KUKA KRL program: MyProgram_008().src

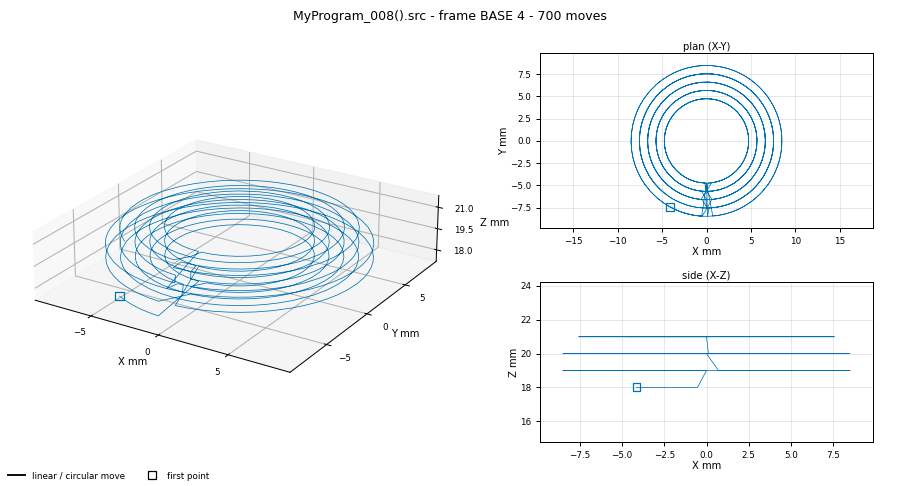
[picture p0: tool path of MyProgram_008().src in frame BASE 4, 700 of 700 moves have a stored position in this frame; points joined in program order, loops and branches not executed]
&ACCESS RVP
&REL 1
&PARAM TEMPLATE = C:\KRC\Roboter\Template\vorgabe
&PARAM EDITMASK = *
DEF MyProgram_008()
; ---- Setting reference (Base) ----
$BASE = BASE_DATA[4]

; --------------------------
; ---- Setting tool (TCP) ----
$TOOL = TOOL_DATA[3]
; --------------------------

$VEL.CP = VEL_APROX_PRINT
Startdeposition()
$VEL.CP = VEL_PRINT
LIN {X -4.1408,Y -7.4105,Z 18,A -3.2305,B 0,C 0,E1 0.1598,E2 90.0712} C_DIS
LIN {X -3.4628,Y -7.7493,Z 18,A -3.22,B 0,C 0,E1 0.1598,E2 90.0712} C_DIS
LIN {X -2.7578,Y -8.0269,Z 18,A -3.2059,B 0,C 0,E1 0.1598,E2 90.0712} C_DIS
LIN {X -2.031,Y -8.2415,Z 18,A -3.1884,B 0,C 0,E1 0.1598,E2 90.0712} C_DIS
LIN {X -1.288,Y -8.391,Z 18,A -3.1675,B 0,C 0,E1 0.1598,E2 90.0713} C_DIS
LIN {X -0.5343,Y -8.4709,Z 18,A -3.1433,B 0,C 0,E1 0.1598,E2 90.0713} C_DIS
LIN {X -0.5343,Y -8.4709,Z 18,A -3.1433,B 0,C 0,E1 0.1598,E2 90.0713} C_DIS
Enddeposition()
LIN {X 0.0003,Y -4.7568,Z 19,A -2.951,B 0,C 0,E1 0.1598,E2 90.0603} C_DIS
Startdeposition()
$VEL.CP = VEL_PRINT
LIN {X 0.0003,Y -4.7568,Z 19,A -2.9567,B 0,C 0,E1 0.1598,E2 90.0661} C_DIS
LIN {X -0.9266,Y -4.6606,Z 19,A -2.9915,B 0,C 0,E1 0.1598,E2 90.0709} C_DIS
LIN {X -1.6437,Y -4.457,Z 19,A -3.0098,B 0,C 0,E1 0.1598,E2 90.0715} C_DIS
LIN {X -2.3205,Y -4.1449,Z 19,A -3.0215,B 0,C 0,E1 0.1598,E2 90.0715} C_DIS
LIN {X -2.9394,Y -3.7297,Z 19,A -3.0266,B 0,C 0,E1 0.1598,E2 90.0715} C_DIS
LIN {X -3.4873,Y -3.2244,Z 19,A -3.0253,B 0,C 0,E1 0.1598,E2 90.0714} C_DIS
LIN {X -3.9485,Y -2.6389,Z 19,A -3.0174,B 0,C 0,E1 0.1598,E2 90.0714} C_DIS
LIN {X -4.314,Y -1.9893,Z 19,A -3.0034,B 0,C 0,E1 0.1598,E2 90.0714} C_DIS
LIN {X -4.5707,Y -1.2895,Z 19,A -2.9832,B 0,C 0,E1 0.1598,E2 90.0714} C_DIS
LIN {X -4.716,Y -0.5586,Z 19,A -2.9577,B 0,C 0,E1 0.1598,E2 90.0714} C_DIS
LIN {X -4.7458,Y 0.1861,Z 19,A -2.9273,B 0,C 0,E1 0.1598,E2 90.0714} C_DIS
LIN {X -4.6607,Y 0.9267,Z 19,A -2.8929,B 0,C 0,E1 0.1598,E2 90.0714} C_DIS
LIN {X -4.4566,Y 1.6437,Z 19,A -2.8551,B 0,C 0,E1 0.1598,E2 90.0715} C_DIS
LIN {X -4.1446,Y 2.3207,Z 19,A -2.8151,B 0,C 0,E1 0.1598,E2 90.0715} C_DIS
LIN {X -3.7315,Y 2.9411,Z 19,A -2.7737,B 0,C 0,E1 0.1598,E2 90.0717} C_DIS
LIN {X -3.225,Y 3.4882,Z 19,A -2.732,B 0,C 0,E1 0.1598,E2 90.0717} C_DIS
LIN {X -2.6388,Y 3.9486,Z 19,A -2.691,B 0,C 0,E1 0.1598,E2 90.0719} C_DIS
LIN {X -1.9887,Y 4.313,Z 19,A -2.6517,B 0,C 0,E1 0.1598,E2 90.0719} C_DIS
LIN {X -1.1995,Y 4.5956,Z 19,A -2.6107,B 0,C 0,E1 0.1598,E2 90.0721} C_DIS
LIN {X -0.5587,Y 4.7185,Z 19,A -2.5819,B 0,C 0,E1 0.1598,E2 90.0721} C_DIS
LIN {X 0.1862,Y 4.749,Z 19,A -2.5532,B 0,C 0,E1 0.1598,E2 90.0721} C_DIS
LIN {X 0.9266,Y 4.6606,Z 19,A -2.5296,B 0,C 0,E1 0.1598,E2 90.0721} C_DIS
LIN {X 1.6433,Y 4.456,Z 19,A -2.5118,B 0,C 0,E1 0.1598,E2 90.0721} C_DIS
LIN {X 2.3206,Y 4.1447,Z 19,A -2.5,B 0,C 0,E1 0.1598,E2 90.0721} C_DIS
LIN {X 2.9416,Y 3.7322,Z 19,A -2.4945,B 0,C 0,E1 0.1598,E2 90.0721} C_DIS
LIN {X 3.4881,Y 3.2248,Z 19,A -2.4958,B 0,C 0,E1 0.1598,E2 90.0721} C_DIS
LIN {X 3.9509,Y 2.6404,Z 19,A -2.5035,B 0,C 0,E1 0.1598,E2 90.0721} C_DIS
LIN {X 4.3138,Y 1.989,Z 19,A -2.5177,B 0,C 0,E1 0.1598,E2 90.072} C_DIS
LIN {X 4.5707,Y 1.2894,Z 19,A -2.5379,B 0,C 0,E1 0.1598,E2 90.072} C_DIS
LIN {X 4.7184,Y 0.5588,Z 19,A -2.5635,B 0,C 0,E1 0.1598,E2 90.0719} C_DIS
LIN {X 4.7489,Y -0.1862,Z 19,A -2.594,B 0,C 0,E1 0.1598,E2 90.0719} C_DIS
LIN {X 4.6591,Y -0.9263,Z 19,A -2.6287,B 0,C 0,E1 0.1598,E2 90.0718} C_DIS
LIN {X 4.4556,Y -1.6435,Z 19,A -2.6666,B 0,C 0,E1 0.1598,E2 90.0718} C_DIS
LIN {X 4.1448,Y -2.3207,Z 19,A -2.7068,B 0,C 0,E1 0.1598,E2 90.0718} C_DIS
LIN {X 3.7299,Y -2.9399,Z 19,A -2.7484,B 0,C 0,E1 0.1598,E2 90.0718} C_DIS
LIN {X 3.2242,Y -3.4874,Z 19,A -2.7903,B 0,C 0,E1 0.1598,E2 90.0718} C_DIS
LIN {X 2.6388,Y -3.9486,Z 19,A -2.8314,B 0,C 0,E1 0.1598,E2 90.0717} C_DIS
LIN {X 1.9887,Y -4.313,Z 19,A -2.8708,B 0,C 0,E1 0.1598,E2 90.0717} C_DIS
LIN {X 1.1996,Y -4.5956,Z 19,A -2.9118,B 0,C 0,E1 0.1598,E2 90.0717} C_DIS
LIN {X 0.5588,Y -4.7187,Z 19,A -2.9405,B 0,C 0,E1 0.1598,E2 90.0717} C_DIS
LIN {X 0.5588,Y -4.7187,Z 19,A -2.9405,B 0,C 0,E1 0.1598,E2 90.0717} C_DIS
Enddeposition()
LIN {X 0,Y -5.6862,Z 19,A -3.001,B 0,C 0,E1 0.1598,E2 90.0704} C_DIS
Startdeposition()
$VEL.CP = VEL_PRINT
LIN {X 0.6409,Y -5.6452,Z 19,A -2.9769,B 0,C 0,E1 0.1598,E2 90.0715} C_DIS
LIN {X 1.4817,Y -5.4861,Z 19,A -2.9393,B 0,C 0,E1 0.1598,E2 90.0716} C_DIS
LIN {X 2.2884,Y -5.2009,Z 19,A -2.8976,B 0,C 0,E1 0.1598,E2 90.0716} C_DIS
LIN {X 3.0434,Y -4.7981,Z 19,A -2.8527,B 0,C 0,E1 0.1598,E2 90.0716} C_DIS
LIN {X 3.7291,Y -4.2862,Z 19,A -2.8058,B 0,C 0,E1 0.1598,E2 90.0717} C_DIS
LIN {X 4.3305,Y -3.6775,Z 19,A -2.7578,B 0,C 0,E1 0.1598,E2 90.0717} C_DIS
LIN {X 4.8347,Y -2.986,Z 19,A -2.7098,B 0,C 0,E1 0.1598,E2 90.0717} C_DIS
LIN {X 5.2278,Y -2.226,Z 19,A -2.663,B 0,C 0,E1 0.1598,E2 90.0717} C_DIS
LIN {X 5.5023,Y -1.4156,Z 19,A -2.6184,B 0,C 0,E1 0.1598,E2 90.0717} C_DIS
LIN {X 5.6534,Y -0.5733,Z 19,A -2.5771,B 0,C 0,E1 0.1598,E2 90.0717} C_DIS
LIN {X 5.6763,Y 0.2822,Z 19,A -2.5399,B 0,C 0,E1 0.1598,E2 90.0717} C_DIS
LIN {X 5.5702,Y 1.1315,Z 19,A -2.5077,B 0,C 0,E1 0.1598,E2 90.0718} C_DIS
LIN {X 5.3355,Y 1.9546,Z 19,A -2.4814,B 0,C 0,E1 0.1598,E2 90.0718} C_DIS
LIN {X 4.9812,Y 2.7335,Z 19,A -2.4614,B 0,C 0,E1 0.1598,E2 90.0719} C_DIS
LIN {X 4.514,Y 3.4505,Z 19,A -2.4483,B 0,C 0,E1 0.1598,E2 90.072} C_DIS
LIN {X 3.945,Y 4.0897,Z 19,A -2.4422,B 0,C 0,E1 0.1598,E2 90.072} C_DIS
LIN {X 3.2863,Y 4.6361,Z 19,A -2.4434,B 0,C 0,E1 0.1598,E2 90.0721} C_DIS
LIN {X 2.5533,Y 5.0782,Z 19,A -2.4518,B 0,C 0,E1 0.1598,E2 90.0721} C_DIS
LIN {X 1.7619,Y 5.4046,Z 19,A -2.4672,B 0,C 0,E1 0.1598,E2 90.0722} C_DIS
LIN {X 0.9303,Y 5.6086,Z 19,A -2.4893,B 0,C 0,E1 0.1598,E2 90.0722} C_DIS
LIN {X 0.0776,Y 5.6849,Z 19,A -2.5175,B 0,C 0,E1 0.1598,E2 90.0722} C_DIS
LIN {X -0.7768,Y 5.6314,Z 19,A -2.5513,B 0,C 0,E1 0.1598,E2 90.0722} C_DIS
LIN {X -1.614,Y 5.4516,Z 19,A -2.5898,B 0,C 0,E1 0.1598,E2 90.0722} C_DIS
LIN {X -2.4546,Y 5.1327,Z 19,A -2.6342,B 0,C 0,E1 0.1598,E2 90.072} C_DIS
LIN {X -3.5239,Y 4.4596,Z 19,A -2.7019,B 0,C 0,E1 0.1598,E2 90.0718} C_DIS
LIN {X -4.0794,Y 3.9571,Z 19,A -2.7436,B 0,C 0,E1 0.1598,E2 90.0718} C_DIS
LIN {X -4.5642,Y 3.3862,Z 19,A -2.7855,B 0,C 0,E1 0.1598,E2 90.0717} C_DIS
LIN {X -4.9699,Y 2.7566,Z 19,A -2.827,B 0,C 0,E1 0.1598,E2 90.0717} C_DIS
LIN {X -5.2905,Y 2.0796,Z 19,A -2.8673,B 0,C 0,E1 0.1598,E2 90.0715} C_DIS
LIN {X -5.5194,Y 1.3661,Z 19,A -2.9058,B 0,C 0,E1 0.1598,E2 90.0715} C_DIS
LIN {X -5.6499,Y 0.6283,Z 19,A -2.9417,B 0,C 0,E1 0.1598,E2 90.0714} C_DIS
LIN {X -5.6842,Y -0.12,Z 19,A -2.9746,B 0,C 0,E1 0.1598,E2 90.0714} C_DIS
LIN {X -5.6165,Y -0.8662,Z 19,A -3.0036,B 0,C 0,E1 0.1598,E2 90.0713} C_DIS
LIN {X -5.4547,Y -1.5974,Z 19,A -3.0285,B 0,C 0,E1 0.1598,E2 90.0713} C_DIS
LIN {X -5.1973,Y -2.3009,Z 19,A -3.0488,B 0,C 0,E1 0.1598,E2 90.0713} C_DIS
LIN {X -4.8517,Y -2.9656,Z 19,A -3.0642,B 0,C 0,E1 0.1598,E2 90.0713} C_DIS
LIN {X -4.4183,Y -3.5769,Z 19,A -3.0741,B 0,C 0,E1 0.1598,E2 90.0713} C_DIS
LIN {X -3.9082,Y -4.1255,Z 19,A -3.0786,B 0,C 0,E1 0.1598,E2 90.0713} C_DIS
LIN {X -3.3325,Y -4.6046,Z 19,A -3.0778,B 0,C 0,E1 0.1598,E2 90.0713} C_DIS
LIN {X -2.6973,Y -5.0015,Z 19,A -3.0713,B 0,C 0,E1 0.1598,E2 90.0713} C_DIS
LIN {X -2.0167,Y -5.3143,Z 19,A -3.0596,B 0,C 0,E1 0.1598,E2 90.0714} C_DIS
LIN {X -1.3007,Y -5.5351,Z 19,A -3.0427,B 0,C 0,E1 0.1598,E2 90.0714} C_DIS
LIN {X -0.5612,Y -5.6557,Z 19,A -3.0207,B 0,C 0,E1 0.1598,E2 90.0715} C_DIS
LIN {X -0.5612,Y -5.6557,Z 19,A -3.0207,B 0,C 0,E1 0.1598,E2 90.0715} C_DIS
Enddeposition()
LIN {X 0.0261,Y -6.6218,Z 19,A -3.0391,B 0,C 0,E1 0.1598,E2 90.0703} C_DIS
Startdeposition()
$VEL.CP = VEL_PRINT
LIN {X -0.8856,Y -6.5586,Z 19,A -3.0709,B 0,C 0,E1 0.1598,E2 90.0714} C_DIS
LIN {X -1.6037,Y -6.4211,Z 19,A -3.0915,B 0,C 0,E1 0.1598,E2 90.0714} C_DIS
LIN {X -2.3028,Y -6.2069,Z 19,A -3.1081,B 0,C 0,E1 0.1598,E2 90.0714} C_DIS
LIN {X -2.9723,Y -5.9126,Z 19,A -3.1201,B 0,C 0,E1 0.1598,E2 90.0714} C_DIS
LIN {X -3.607,Y -5.5497,Z 19,A -3.1281,B 0,C 0,E1 0.1598,E2 90.0714} C_DIS
LIN {X -4.1979,Y -5.1188,Z 19,A -3.1315,B 0,C 0,E1 0.1598,E2 90.0713} C_DIS
LIN {X -4.7363,Y -4.6238,Z 19,A -3.1303,B 0,C 0,E1 0.1598,E2 90.0713} C_DIS
LIN {X -5.217,Y -4.0727,Z 19,A -3.1246,B 0,C 0,E1 0.1598,E2 90.0713} C_DIS
LIN {X -5.6344,Y -3.4723,Z 19,A -3.1145,B 0,C 0,E1 0.1598,E2 90.0713} C_DIS
LIN {X -5.9829,Y -2.8295,Z 19,A -3.1002,B 0,C 0,E1 0.1598,E2 90.0713} C_DIS
LIN {X -6.2578,Y -2.1521,Z 19,A -3.0817,B 0,C 0,E1 0.1598,E2 90.0713} C_DIS
LIN {X -6.4587,Y -1.449,Z 19,A -3.0593,B 0,C 0,E1 0.1598,E2 90.0713} C_DIS
LIN {X -6.5806,Y -0.7279,Z 19,A -3.0334,B 0,C 0,E1 0.1598,E2 90.0713} C_DIS
LIN {X -6.6194,Y 0.0024,Z 19,A -3.004,B 0,C 0,E1 0.1598,E2 90.0713} C_DIS
LIN {X -6.5797,Y 0.7325,Z 19,A -2.9717,B 0,C 0,E1 0.1598,E2 90.0713} C_DIS
LIN {X -6.4575,Y 1.4535,Z 19,A -2.9368,B 0,C 0,E1 0.1598,E2 90.0713} C_DIS
LIN {X -6.2582,Y 2.1571,Z 19,A -2.8999,B 0,C 0,E1 0.1598,E2 90.0715} C_DIS
LIN {X -5.9836,Y 2.8348,Z 19,A -2.8612,B 0,C 0,E1 0.1598,E2 90.0715} C_DIS
LIN {X -5.6316,Y 3.4757,Z 19,A -2.8212,B 0,C 0,E1 0.1598,E2 90.0716} C_DIS
LIN {X -5.2138,Y 4.0758,Z 19,A -2.7805,B 0,C 0,E1 0.1598,E2 90.0716} C_DIS
LIN {X -4.7331,Y 4.6268,Z 19,A -2.7396,B 0,C 0,E1 0.1598,E2 90.0718} C_DIS
LIN {X -4.195,Y 5.1216,Z 19,A -2.6989,B 0,C 0,E1 0.1598,E2 90.0718} C_DIS
LIN {X -3.6043,Y 5.5527,Z 19,A -2.659,B 0,C 0,E1 0.1598,E2 90.0719} C_DIS
LIN {X -2.97,Y 5.9168,Z 19,A -2.6202,B 0,C 0,E1 0.1598,E2 90.072} C_DIS
LIN {X -2.2998,Y 6.2097,Z 19,A -2.5832,B 0,C 0,E1 0.1598,E2 90.072} C_DIS
LIN {X -1.6007,Y 6.4242,Z 19,A -2.5483,B 0,C 0,E1 0.1598,E2 90.0722} C_DIS
LIN {X -0.701,Y 6.5862,Z 19,A -2.5083,B 0,C 0,E1 0.1598,E2 90.0722} C_DIS
LIN {X 0.455,Y 6.6038,Z 19,A -2.4649,B 0,C 0,E1 0.1598,E2 90.0722} C_DIS
LIN {X 1.6036,Y 6.4264,Z 19,A -2.43,B 0,C 0,E1 0.1598,E2 90.0723} C_DIS
LIN {X 2.5114,Y 6.1237,Z 19,A -2.4093,B 0,C 0,E1 0.1598,E2 90.0723} C_DIS
LIN {X 3.2013,Y 5.7918,Z 19,A -2.3979,B 0,C 0,E1 0.1598,E2 90.0723} C_DIS
LIN {X 3.849,Y 5.3838,Z 19,A -2.3913,B 0,C 0,E1 0.1598,E2 90.0723} C_DIS
LIN {X 4.4444,Y 4.9029,Z 19,A -2.3896,B 0,C 0,E1 0.1598,E2 90.0723} C_DIS
LIN {X 4.9809,Y 4.357,Z 19,A -2.393,B 0,C 0,E1 0.1598,E2 90.0722} C_DIS
LIN {X 5.4509,Y 3.7528,Z 19,A -2.4012,B 0,C 0,E1 0.1598,E2 90.0722} C_DIS
LIN {X 5.8483,Y 3.0985,Z 19,A -2.4143,B 0,C 0,E1 0.1598,E2 90.0721} C_DIS
LIN {X 6.1677,Y 2.4028,Z 19,A -2.4321,B 0,C 0,E1 0.1598,E2 90.0721} C_DIS
LIN {X 6.4042,Y 1.6746,Z 19,A -2.4542,B 0,C 0,E1 0.1598,E2 90.072} C_DIS
LIN {X 6.5537,Y 0.9237,Z 19,A -2.4806,B 0,C 0,E1 0.1598,E2 90.072} C_DIS
LIN {X 6.6156,Y 0.1609,Z 19,A -2.5107,B 0,C 0,E1 0.1598,E2 90.0719} C_DIS
LIN {X 6.5914,Y -0.6042,Z 19,A -2.5441,B 0,C 0,E1 0.1598,E2 90.0719} C_DIS
LIN {X 6.4774,Y -1.3612,Z 19,A -2.5805,B 0,C 0,E1 0.1598,E2 90.0719} C_DIS
LIN {X 6.2764,Y -2.0999,Z 19,A -2.6193,B 0,C 0,E1 0.1598,E2 90.0718} C_DIS
LIN {X 5.9941,Y -2.8114,Z 19,A -2.66,B 0,C 0,E1 0.1598,E2 90.0718} C_DIS
LIN {X 5.6304,Y -3.4851,Z 19,A -2.702,B 0,C 0,E1 0.1598,E2 90.0718} C_DIS
LIN {X 5.1873,Y -4.1094,Z 19,A -2.7448,B 0,C 0,E1 0.1598,E2 90.0718} C_DIS
LIN {X 4.6785,Y -4.6812,Z 19,A -2.7878,B 0,C 0,E1 0.1598,E2 90.0717} C_DIS
LIN {X 4.1066,Y -5.19,Z 19,A -2.8305,B 0,C 0,E1 0.1598,E2 90.0717} C_DIS
LIN {X 3.4797,Y -5.6294,Z 19,A -2.8722,B 0,C 0,E1 0.1598,E2 90.0717} C_DIS
LIN {X 2.8072,Y -5.9951,Z 19,A -2.9124,B 0,C 0,E1 0.1598,E2 90.0717} C_DIS
LIN {X 2.0961,Y -6.2792,Z 19,A -2.9506,B 0,C 0,E1 0.1598,E2 90.0717} C_DIS
LIN {X 1.3572,Y -6.4796,Z 19,A -2.9862,B 0,C 0,E1 0.1598,E2 90.0716} C_DIS
LIN {X 0.5998,Y -6.5922,Z 19,A -3.0188,B 0,C 0,E1 0.1598,E2 90.0716} C_DIS
LIN {X 0.5998,Y -6.5922,Z 19,A -3.0188,B 0,C 0,E1 0.1598,E2 90.0716} C_DIS
Enddeposition()
LIN {X 0.0596,Y -7.5563,Z 19,A -3.0785,B 0,C 0,E1 0.1598,E2 90.0703} C_DIS
Startdeposition()
$VEL.CP = VEL_PRINT
LIN {X 0.9093,Y -7.5022,Z 19,A -3.0462,B 0,C 0,E1 0.1598,E2 90.0715} C_DIS
LIN {X 2.0403,Y -7.2731,Z 19,A -2.995,B 0,C 0,E1 0.1598,E2 90.0715} C_DIS
LIN {X 2.9949,Y -6.9378,Z 19,A -2.9457,B 0,C 0,E1 0.1598,E2 90.0715} C_DIS
LIN {X 3.9106,Y -6.4663,Z 19,A -2.8921,B 0,C 0,E1 0.1598,E2 90.0716} C_DIS
LIN {X 4.6992,Y -5.9141,Z 19,A -2.8396,B 0,C 0,E1 0.1598,E2 90.0716} C_DIS
LIN {X 5.276,Y -5.4037,Z 19,A -2.7968,B 0,C 0,E1 0.1598,E2 90.0717} C_DIS
LIN {X 5.7989,Y -4.8384,Z 19,A -2.7535,B 0,C 0,E1 0.1598,E2 90.0717} C_DIS
LIN {X 6.3712,Y -4.0643,Z 19,A -2.6994,B 0,C 0,E1 0.1598,E2 90.0717} C_DIS
LIN {X 7.0456,Y -2.735,Z 19,A -2.6176,B 0,C 0,E1 0.1598,E2 90.0712} C_DIS
LIN {X 7.3713,Y -1.6678,Z 19,A -2.5604,B 0,C 0,E1 0.1598,E2 90.0715} C_DIS
LIN {X 7.5325,Y -0.6167,Z 19,A -2.5098,B 0,C 0,E1 0.1598,E2 90.0716} C_DIS
LIN {X 7.5419,Y 0.4018,Z 19,A -2.4662,B 0,C 0,E1 0.1598,E2 90.0717} C_DIS
LIN {X 7.4027,Y 1.5186,Z 19,A -2.4237,B 0,C 0,E1 0.1598,E2 90.0717} C_DIS
LIN {X 7.1897,Y 2.3275,Z 19,A -2.3975,B 0,C 0,E1 0.1598,E2 90.072} C_DIS
LIN {X 6.7449,Y 3.4003,Z 19,A -2.368,B 0,C 0,E1 0.1598,E2 90.0717} C_DIS
LIN {X 6.342,Y 4.1018,Z 19,A -2.3534,B 0,C 0,E1 0.1598,E2 90.0721} C_DIS
LIN {X 5.8671,Y 4.7568,Z 19,A -2.3432,B 0,C 0,E1 0.1598,E2 90.0721} C_DIS
LIN {X 5.3248,Y 5.3573,Z 19,A -2.3378,B 0,C 0,E1 0.1598,E2 90.0722} C_DIS
LIN {X 4.5636,Y 6.023,Z 19,A -2.3375,B 0,C 0,E1 0.1598,E2 90.0722} C_DIS
LIN {X 3.61,Y 6.635,Z 19,A -2.3468,B 0,C 0,E1 0.1598,E2 90.0722} C_DIS
LIN {X 2.6664,Y 7.0708,Z 19,A -2.3633,B 0,C 0,E1 0.1598,E2 90.0722} C_DIS
LIN {X 1.6408,Y 7.377,Z 19,A -2.3883,B 0,C 0,E1 0.1598,E2 90.0723} C_DIS
LIN {X 0.7499,Y 7.5202,Z 19,A -2.4152,B 0,C 0,E1 0.1598,E2 90.0723} C_DIS
LIN {X -0.2197,Y 7.5539,Z 19,A -2.4496,B 0,C 0,E1 0.1598,E2 90.0723} C_DIS
LIN {X -1.2608,Y 7.4511,Z 19,A -2.4923,B 0,C 0,E1 0.1598,E2 90.0723} C_DIS
LIN {X -2.3419,Y 7.1807,Z 19,A -2.5436,B 0,C 0,E1 0.1598,E2 90.0722} C_DIS
LIN {X -3.1716,Y 6.8543,Z 19,A -2.588,B 0,C 0,E1 0.1598,E2 90.0721} C_DIS
LIN {X -3.9585,Y 6.4347,Z 19,A -2.6347,B 0,C 0,E1 0.1598,E2 90.072} C_DIS
LIN {X -4.9384,Y 5.7195,Z 19,A -2.7009,B 0,C 0,E1 0.1598,E2 90.0717} C_DIS
LIN {X -5.6771,Y 4.9879,Z 19,A -2.7589,B 0,C 0,E1 0.1598,E2 90.0717} C_DIS
LIN {X -6.2659,Y 4.2161,Z 19,A -2.8131,B 0,C 0,E1 0.1598,E2 90.0716} C_DIS
LIN {X -6.759,Y 3.38,Z 19,A -2.8664,B 0,C 0,E1 0.1598,E2 90.0713} C_DIS
LIN {X -7.2749,Y 2.0498,Z 19,A -2.9409,B 0,C 0,E1 0.1598,E2 90.0707} C_DIS
LIN {X -7.5164,Y 0.7835,Z 19,A -3.0033,B 0,C 0,E1 0.1598,E2 90.0707} C_DIS
LIN {X -7.5569,Y -0.0876,Z 19,A -3.0419,B 0,C 0,E1 0.1598,E2 90.0711} C_DIS
LIN {X -7.4292,Y -1.3623,Z 19,A -3.0904,B 0,C 0,E1 0.1598,E2 90.0706} C_DIS
LIN {X -7.2654,Y -2.0847,Z 19,A -3.1154,B 0,C 0,E1 0.1598,E2 90.071} C_DIS
LIN {X -6.861,Y -3.158,Z 19,A -3.1457,B 0,C 0,E1 0.1598,E2 90.0708} C_DIS
LIN {X -6.2752,Y -4.2109,Z 19,A -3.1686,B 0,C 0,E1 0.1598,E2 90.0708} C_DIS
LIN {X -5.7777,Y -4.8704,Z 19,A -3.1784,B 0,C 0,E1 0.1598,E2 90.071} C_DIS
LIN {X -5.079,Y -5.5909,Z 19,A -3.1833,B 0,C 0,E1 0.1598,E2 90.071} C_DIS
LIN {X -4.4563,Y -6.0978,Z 19,A -3.182,B 0,C 0,E1 0.1598,E2 90.0712} C_DIS
LIN {X -3.7835,Y -6.5358,Z 19,A -3.1759,B 0,C 0,E1 0.1598,E2 90.0712} C_DIS
LIN {X -3.0689,Y -6.9019,Z 19,A -3.1652,B 0,C 0,E1 0.1598,E2 90.0712} C_DIS
LIN {X -1.9814,Y -7.2927,Z 19,A -3.1418,B 0,C 0,E1 0.1598,E2 90.0713} C_DIS
LIN {X -0.9532,Y -7.4972,Z 19,A -3.1129,B 0,C 0,E1 0.1598,E2 90.0713} C_DIS
LIN {X 0.0596,Y -7.5563,Z 19,A -3.0782,B 0,C 0,E1 0.1598,E2 90.0715} C_DIS
Enddeposition()
LIN {X 0.0596,Y -7.5563,Z 19,A -3.0782,B 0,C 0,E1 0.1598,E2 90.0715} C_DIS
Startdeposition()
$VEL.CP = VEL_PRINT
LIN {X -0.4894,Y -8.4742,Z 19,A -3.137,B 0,C 0,E1 0.1598,E2 90.0708} C_DIS
LIN {X -1.2506,Y -8.3958,Z 19,A -3.162,B 0,C 0,E1 0.1598,E2 90.0713} C_DIS
LIN {X -2.0013,Y -8.2484,Z 19,A -3.1833,B 0,C 0,E1 0.1598,E2 90.0713} C_DIS
LIN {X -2.7359,Y -8.0344,Z 19,A -3.2012,B 0,C 0,E1 0.1598,E2 90.0713} C_DIS
LIN {X -3.4483,Y -7.7557,Z 19,A -3.2155,B 0,C 0,E1 0.1598,E2 90.0713} C_DIS
LIN {X -4.1333,Y -7.4148,Z 19,A -3.2261,B 0,C 0,E1 0.1598,E2 90.0713} C_DIS
LIN {X -4.7837,Y -7.0118,Z 19,A -3.2329,B 0,C 0,E1 0.1598,E2 90.0712} C_DIS
LIN {X -5.5434,Y -6.4306,Z 19,A -3.2361,B 0,C 0,E1 0.1598,E2 90.071} C_DIS
LIN {X -6.3513,Y -5.6359,Z 19,A -3.232,B 0,C 0,E1 0.1598,E2 90.071} C_DIS
LIN {X -6.9717,Y -4.8405,Z 19,A -3.2212,B 0,C 0,E1 0.1598,E2 90.071} C_DIS
LIN {X -7.3989,Y -4.1558,Z 19,A -3.208,B 0,C 0,E1 0.1598,E2 90.071} C_DIS
LIN {X -7.7607,Y -3.4345,Z 19,A -3.1909,B 0,C 0,E1 0.1598,E2 90.071} C_DIS
LIN {X -8.0526,Y -2.682,Z 19,A -3.1698,B 0,C 0,E1 0.1598,E2 90.071} C_DIS
LIN {X -8.2711,Y -1.905,Z 19,A -3.1451,B 0,C 0,E1 0.1598,E2 90.071} C_DIS
LIN {X -8.4144,Y -1.1108,Z 19,A -3.1168,B 0,C 0,E1 0.1598,E2 90.071} C_DIS
LIN {X -8.4903,Y -0.1049,Z 19,A -3.077,B 0,C 0,E1 0.1598,E2 90.0709} C_DIS
LIN {X -8.4259,Y 1.0155,Z 19,A -3.0273,B 0,C 0,E1 0.1598,E2 90.0709} C_DIS
LIN {X -8.2936,Y 1.8064,Z 19,A -2.9895,B 0,C 0,E1 0.1598,E2 90.0713} C_DIS
LIN {X -8.0861,Y 2.581,Z 19,A -2.9492,B 0,C 0,E1 0.1598,E2 90.0713} C_DIS
LIN {X -7.8078,Y 3.3331,Z 19,A -2.9073,B 0,C 0,E1 0.1598,E2 90.0714} C_DIS
LIN {X -7.4578,Y 4.0548,Z 19,A -2.864,B 0,C 0,E1 0.1598,E2 90.0714} C_DIS
LIN {X -7.041,Y 4.7398,Z 19,A -2.8198,B 0,C 0,E1 0.1598,E2 90.0716} C_DIS
LIN {X -6.4349,Y 5.5383,Z 19,A -2.7637,B 0,C 0,E1 0.1598,E2 90.0716} C_DIS
LIN {X -5.6183,Y 6.3622,Z 19,A -2.6989,B 0,C 0,E1 0.1598,E2 90.0716} C_DIS
LIN {X -4.9802,Y 6.8722,Z 19,A -2.6541,B 0,C 0,E1 0.1598,E2 90.0719} C_DIS
LIN {X -4.2961,Y 7.3187,Z 19,A -2.61,B 0,C 0,E1 0.1598,E2 90.0719} C_DIS
LIN {X -3.5723,Y 7.6974,Z 19,A -2.5674,B 0,C 0,E1 0.1598,E2 90.0721} C_DIS
LIN {X -2.8157,Y 8.005,Z 19,A -2.5265,B 0,C 0,E1 0.1598,E2 90.0721} C_DIS
LIN {X -2.033,Y 8.2385,Z 19,A -2.4878,B 0,C 0,E1 0.1598,E2 90.0722} C_DIS
LIN {X -1.2315,Y 8.396,Z 19,A -2.4515,B 0,C 0,E1 0.1598,E2 90.0722} C_DIS
LIN {X -0.4187,Y 8.4762,Z 19,A -2.4181,B 0,C 0,E1 0.1598,E2 90.0723} C_DIS
LIN {X 0.6022,Y 8.4692,Z 19,A -2.3807,B 0,C 0,E1 0.1598,E2 90.0723} C_DIS
LIN {X 1.7078,Y 8.3157,Z 19,A -2.3464,B 0,C 0,E1 0.1598,E2 90.0724} C_DIS
LIN {X 2.5031,Y 8.1114,Z 19,A -2.3256,B 0,C 0,E1 0.1598,E2 90.0724} C_DIS
LIN {X 3.2749,Y 7.8313,Z 19,A -2.309,B 0,C 0,E1 0.1598,E2 90.0724} C_DIS
LIN {X 4.016,Y 7.4779,Z 19,A -2.2965,B 0,C 0,E1 0.1598,E2 90.0724} C_DIS
LIN {X 4.7194,Y 7.0545,Z 19,A -2.2885,B 0,C 0,E1 0.1598,E2 90.0724} C_DIS
LIN {X 5.5379,Y 6.4353,Z 19,A -2.2844,B 0,C 0,E1 0.1598,E2 90.0722} C_DIS
LIN {X 6.3767,Y 5.6023,Z 19,A -2.2886,B 0,C 0,E1 0.1598,E2 90.0721} C_DIS
LIN {X 6.8766,Y 4.9827,Z 19,A -2.2965,B 0,C 0,E1 0.1598,E2 90.0721} C_DIS
LIN {X 7.414,Y 4.1342,Z 19,A -2.3127,B 0,C 0,E1 0.1598,E2 90.0721} C_DIS
LIN {X 7.7694,Y 3.4136,Z 19,A -2.3303,B 0,C 0,E1 0.1598,E2 90.0721} C_DIS
LIN {X 8.0582,Y 2.6638,Z 19,A -2.3515,B 0,C 0,E1 0.1598,E2 90.0721} C_DIS
LIN {X 8.2747,Y 1.89,Z 19,A -2.3764,B 0,C 0,E1 0.1598,E2 90.0721} C_DIS
LIN {X 8.4161,Y 1.099,Z 19,A -2.4048,B 0,C 0,E1 0.1598,E2 90.0721} C_DIS
LIN {X 8.4905,Y 0.0975,Z 19,A -2.4444,B 0,C 0,E1 0.1598,E2 90.0717} C_DIS
LIN {X 8.4112,Y -1.1261,Z 19,A -2.4991,B 0,C 0,E1 0.1598,E2 90.0714} C_DIS
LIN {X 8.2559,Y -1.9647,Z 19,A -2.5409,B 0,C 0,E1 0.1598,E2 90.0718} C_DIS
LIN {X 8.0176,Y -2.7835,Z 19,A -2.5846,B 0,C 0,E1 0.1598,E2 90.0718} C_DIS
LIN {X 7.698,Y -3.5741,Z 19,A -2.63,B 0,C 0,E1 0.1598,E2 90.0718} C_DIS
LIN {X 7.3003,Y -4.3286,Z 19,A -2.6767,B 0,C 0,E1 0.1598,E2 90.0718} C_DIS
LIN {X 6.8291,Y -5.0396,Z 19,A -2.7243,B 0,C 0,E1 0.1598,E2 90.0717} C_DIS
LIN {X 6.0607,Y -5.947,Z 19,A -2.791,B 0,C 0,E1 0.1598,E2 90.0715} C_DIS
LIN {X 5.2855,Y -6.6411,Z 19,A -2.8491,B 0,C 0,E1 0.1598,E2 90.0715} C_DIS
LIN {X 4.6093,Y -7.1265,Z 19,A -2.8947,B 0,C 0,E1 0.1598,E2 90.0715} C_DIS
LIN {X 3.8888,Y -7.5435,Z 19,A -2.9388,B 0,C 0,E1 0.1598,E2 90.0715} C_DIS
LIN {X 3.1311,Y -7.8881,Z 19,A -2.9813,B 0,C 0,E1 0.1598,E2 90.0715} C_DIS
LIN {X 2.3433,Y -8.1568,Z 19,A -3.0216,B 0,C 0,E1 0.1598,E2 90.0715} C_DIS
LIN {X 1.533,Y -8.3472,Z 19,A -3.0594,B 0,C 0,E1 0.1598,E2 90.0715} C_DIS
LIN {X 0.708,Y -8.4578,Z 19,A -3.0943,B 0,C 0,E1 0.1598,E2 90.0715} C_DIS
LIN {X 0.708,Y -8.4578,Z 19,A -3.0943,B 0,C 0,E1 0.1598,E2 90.0715} C_DIS
Enddeposition()
LIN {X 0.0003,Y -4.7568,Z 20,A -2.9482,B 0,C 0,E1 0.1598,E2 90.0603} C_DIS
Startdeposition()
$VEL.CP = VEL_PRINT
LIN {X 0.0003,Y -4.7568,Z 20,A -2.9539,B 0,C 0,E1 0.1598,E2 90.0661} C_DIS
LIN {X 0.5731,Y -4.7172,Z 20,A -2.936,B 0,C 0,E1 0.1598,E2 90.071} C_DIS
LIN {X 1.3219,Y -4.5623,Z 20,A -2.9026,B 0,C 0,E1 0.1598,E2 90.0717} C_DIS
LIN {X 2.0363,Y -4.2907,Z 20,A -2.8648,B 0,C 0,E1 0.1598,E2 90.0717} C_DIS
LIN {X 2.6983,Y -3.9083,Z 20,A -2.8243,B 0,C 0,E1 0.1598,E2 90.0717} C_DIS
LIN {X 3.2914,Y -3.4262,Z 20,A -2.782,B 0,C 0,E1 0.1598,E2 90.0717} C_DIS
LIN {X 3.7985,Y -2.8538,Z 20,A -2.739,B 0,C 0,E1 0.1598,E2 90.0717} C_DIS
LIN {X 4.2059,Y -2.2068,Z 20,A -2.6965,B 0,C 0,E1 0.1598,E2 90.0717} C_DIS
LIN {X 4.5044,Y -1.5033,Z 20,A -2.6556,B 0,C 0,E1 0.1598,E2 90.0717} C_DIS
LIN {X 4.687,Y -0.7611,Z 20,A -2.6173,B 0,C 0,E1 0.1598,E2 90.0717} C_DIS
LIN {X 4.75,Y 0.0005,Z 20,A -2.5827,B 0,C 0,E1 0.1598,E2 90.0718} C_DIS
LIN {X 4.687,Y 0.762,Z 20,A -2.5526,B 0,C 0,E1 0.1598,E2 90.0718} C_DIS
LIN {X 4.5042,Y 1.5041,Z 20,A -2.5279,B 0,C 0,E1 0.1598,E2 90.0718} C_DIS
LIN {X 4.2058,Y 2.2078,Z 20,A -2.509,B 0,C 0,E1 0.1598,E2 90.0719} C_DIS
LIN {X 3.7984,Y 2.855,Z 20,A -2.4966,B 0,C 0,E1 0.1598,E2 90.0719} C_DIS
LIN {X 3.291,Y 3.4271,Z 20,A -2.4911,B 0,C 0,E1 0.1598,E2 90.0721} C_DIS
LIN {X 2.6981,Y 3.9099,Z 20,A -2.4926,B 0,C 0,E1 0.1598,E2 90.0721} C_DIS
LIN {X 2.0355,Y 4.2913,Z 20,A -2.5009,B 0,C 0,E1 0.1598,E2 90.0721} C_DIS
LIN {X 1.3209,Y 4.5628,Z 20,A -2.5158,B 0,C 0,E1 0.1598,E2 90.0721} C_DIS
LIN {X 0.5719,Y 4.7148,Z 20,A -2.537,B 0,C 0,E1 0.1598,E2 90.0721} C_DIS
LIN {X -0.1918,Y 4.7488,Z 20,A -2.5637,B 0,C 0,E1 0.1598,E2 90.0721} C_DIS
LIN {X -0.9506,Y 4.6545,Z 20,A -2.5957,B 0,C 0,E1 0.1598,E2 90.0721} C_DIS
LIN {X -1.6845,Y 4.4402,Z 20,A -2.6318,B 0,C 0,E1 0.1598,E2 90.0721} C_DIS
LIN {X -2.3746,Y 4.112,Z 20,A -2.671,B 0,C 0,E1 0.1598,E2 90.072} C_DIS
LIN {X -3.0051,Y 3.6797,Z 20,A -2.7125,B 0,C 0,E1 0.1598,E2 90.0719} C_DIS
LIN {X -3.5571,Y 3.1505,Z 20,A -2.7551,B 0,C 0,E1 0.1598,E2 90.0718} C_DIS
LIN {X -4.065,Y 2.4569,Z 20,A -2.803,B 0,C 0,E1 0.1598,E2 90.0716} C_DIS
LIN {X -4.3705,Y 1.8616,Z 20,A -2.8394,B 0,C 0,E1 0.1598,E2 90.0716} C_DIS
LIN {X -4.6135,Y 1.1366,Z 20,A -2.8789,B 0,C 0,E1 0.1598,E2 90.0715} C_DIS
LIN {X -4.7356,Y 0.3817,Z 20,A -2.9153,B 0,C 0,E1 0.1598,E2 90.0714} C_DIS
LIN {X -4.736,Y -0.3828,Z 20,A -2.9476,B 0,C 0,E1 0.1598,E2 90.0714} C_DIS
LIN {X -4.6126,Y -1.1374,Z 20,A -2.9749,B 0,C 0,E1 0.1598,E2 90.0714} C_DIS
LIN {X -4.37,Y -1.8624,Z 20,A -2.9966,B 0,C 0,E1 0.1598,E2 90.0714} C_DIS
LIN {X -4.0134,Y -2.5385,Z 20,A -3.0121,B 0,C 0,E1 0.1598,E2 90.0714} C_DIS
LIN {X -3.5541,Y -3.1493,Z 20,A -3.0211,B 0,C 0,E1 0.1598,E2 90.0714} C_DIS
LIN {X -3.0041,Y -3.6803,Z 20,A -3.0234,B 0,C 0,E1 0.1598,E2 90.0714} C_DIS
LIN {X -2.3737,Y -4.1126,Z 20,A -3.0186,B 0,C 0,E1 0.1598,E2 90.0714} C_DIS
LIN {X -1.6834,Y -4.4405,Z 20,A -3.0072,B 0,C 0,E1 0.1598,E2 90.0715} C_DIS
LIN {X -0.9499,Y -4.6551,Z 20,A -2.9894,B 0,C 0,E1 0.1598,E2 90.0715} C_DIS
LIN {X -0.191,Y -4.7485,Z 20,A -2.9655,B 0,C 0,E1 0.1598,E2 90.0716} C_DIS
LIN {X -0.191,Y -4.7485,Z 20,A -2.9655,B 0,C 0,E1 0.1598,E2 90.0716} C_DIS
Enddeposition()
LIN {X 0.0287,Y -5.6874,Z 20,A -2.9962,B 0,C 0,E1 0.1598,E2 90.0704} C_DIS
Startdeposition()
$VEL.CP = VEL_PRINT
LIN {X -0.8829,Y -5.6139,Z 20,A -3.0276,B 0,C 0,E1 0.1598,E2 90.0715} C_DIS
LIN {X -1.5978,Y -5.4566,Z 20,A -3.0473,B 0,C 0,E1 0.1598,E2 90.0715} C_DIS
LIN {X -2.2849,Y -5.2042,Z 20,A -3.0618,B 0,C 0,E1 0.1598,E2 90.0715} C_DIS
LIN {X -2.9348,Y -4.8676,Z 20,A -3.0713,B 0,C 0,E1 0.1598,E2 90.0715} C_DIS
LIN {X -3.5374,Y -4.4521,Z 20,A -3.0759,B 0,C 0,E1 0.1598,E2 90.0714} C_DIS
LIN {X -4.0791,Y -3.9595,Z 20,A -3.0749,B 0,C 0,E1 0.1598,E2 90.0714} C_DIS
LIN {X -4.5531,Y -3.4018,Z 20,A -3.0687,B 0,C 0,E1 0.1598,E2 90.0714} C_DIS
LIN {X -4.9523,Y -2.7885,Z 20,A -3.0574,B 0,C 0,E1 0.1598,E2 90.0713} C_DIS
LIN {X -5.2716,Y -2.1299,Z 20,A -3.0413,B 0,C 0,E1 0.1598,E2 90.0713} C_DIS
LIN {X -5.5004,Y -1.4345,Z 20,A -3.0203,B 0,C 0,E1 0.1598,E2 90.0713} C_DIS
LIN {X -5.639,Y -0.7159,Z 20,A -2.995,B 0,C 0,E1 0.1598,E2 90.0713} C_DIS
LIN {X -5.6847,Y 0.0147,Z 20,A -2.9658,B 0,C 0,E1 0.1598,E2 90.0713} C_DIS
LIN {X -5.6366,Y 0.7451,Z 20,A -2.9332,B 0,C 0,E1 0.1598,E2 90.0713} C_DIS
LIN {X -5.4925,Y 1.4626,Z 20,A -2.8977,B 0,C 0,E1 0.1598,E2 90.0714} C_DIS
LIN {X -5.2611,Y 2.1572,Z 20,A -2.8599,B 0,C 0,E1 0.1598,E2 90.0715} C_DIS
LIN {X -4.9386,Y 2.8143,Z 20,A -2.8203,B 0,C 0,E1 0.1598,E2 90.0715} C_DIS
LIN {X -4.5354,Y 3.4251,Z 20,A -2.7797,B 0,C 0,E1 0.1598,E2 90.0717} C_DIS
LIN {X -4.0576,Y 3.9795,Z 20,A -2.7387,B 0,C 0,E1 0.1598,E2 90.0717} C_DIS
LIN {X -3.513,Y 4.4683,Z 20,A -2.698,B 0,C 0,E1 0.1598,E2 90.0719} C_DIS
LIN {X -2.4551,Y 5.1324,Z 20,A -2.6309,B 0,C 0,E1 0.1598,E2 90.0719} C_DIS
LIN {X -1.616,Y 5.4509,Z 20,A -2.5867,B 0,C 0,E1 0.1598,E2 90.0721} C_DIS
LIN {X -0.7801,Y 5.6309,Z 20,A -2.5483,B 0,C 0,E1 0.1598,E2 90.0721} C_DIS
LIN {X 0.0731,Y 5.6852,Z 20,A -2.5145,B 0,C 0,E1 0.1598,E2 90.0722} C_DIS
LIN {X 0.9247,Y 5.6092,Z 20,A -2.4863,B 0,C 0,E1 0.1598,E2 90.0722} C_DIS
LIN {X 1.7553,Y 5.4066,Z 20,A -2.4642,B 0,C 0,E1 0.1598,E2 90.0722} C_DIS
LIN {X 2.546,Y 5.0817,Z 20,A -2.4488,B 0,C 0,E1 0.1598,E2 90.0722} C_DIS
LIN {X 3.2786,Y 4.6412,Z 20,A -2.4404,B 0,C 0,E1 0.1598,E2 90.0722} C_DIS
LIN {X 3.9374,Y 4.0967,Z 20,A -2.4391,B 0,C 0,E1 0.1598,E2 90.0722} C_DIS
LIN {X 4.5069,Y 3.4596,Z 20,A -2.4451,B 0,C 0,E1 0.1598,E2 90.0721} C_DIS
LIN {X 4.975,Y 2.7446,Z 20,A -2.4581,B 0,C 0,E1 0.1598,E2 90.072} C_DIS
LIN {X 5.3305,Y 1.9675,Z 20,A -2.4779,B 0,C 0,E1 0.1598,E2 90.072} C_DIS
LIN {X 5.5668,Y 1.1462,Z 20,A -2.5041,B 0,C 0,E1 0.1598,E2 90.0718} C_DIS
LIN {X 5.6751,Y 0.2984,Z 20,A -2.5361,B 0,C 0,E1 0.1598,E2 90.0718} C_DIS
LIN {X 5.6549,Y -0.5559,Z 20,A -2.5731,B 0,C 0,E1 0.1598,E2 90.0718} C_DIS
LIN {X 5.5076,Y -1.3977,Z 20,A -2.6143,B 0,C 0,E1 0.1598,E2 90.0718} C_DIS
LIN {X 5.2356,Y -2.2079,Z 20,A -2.6587,B 0,C 0,E1 0.1598,E2 90.0717} C_DIS
LIN {X 4.8449,Y -2.9679,Z 20,A -2.7054,B 0,C 0,E1 0.1598,E2 90.0717} C_DIS
LIN {X 4.3465,Y -3.6621,Z 20,A -2.7533,B 0,C 0,E1 0.1598,E2 90.0717} C_DIS
LIN {X 3.7488,Y -4.2734,Z 20,A -2.8012,B 0,C 0,E1 0.1598,E2 90.0717} C_DIS
LIN {X 3.0655,Y -4.7874,Z 20,A -2.8482,B 0,C 0,E1 0.1598,E2 90.0717} C_DIS
LIN {X 2.3132,Y -5.1934,Z 20,A -2.8931,B 0,C 0,E1 0.1598,E2 90.0717} C_DIS
LIN {X 1.508,Y -5.4807,Z 20,A -2.9349,B 0,C 0,E1 0.1598,E2 90.0717} C_DIS
LIN {X 0.6689,Y -5.6444,Z 20,A -2.9727,B 0,C 0,E1 0.1598,E2 90.0717} C_DIS
LIN {X 0.0287,Y -5.6874,Z 20,A -2.998,B 0,C 0,E1 0.1598,E2 90.0716} C_DIS
Enddeposition()
LIN {X 0.0287,Y -5.6874,Z 20,A -2.998,B 0,C 0,E1 0.1598,E2 90.0716} C_DIS
Startdeposition()
$VEL.CP = VEL_PRINT
LIN {X 0.6169,Y -6.5912,Z 20,A -3.0143,B 0,C 0,E1 0.1598,E2 90.071} C_DIS
LIN {X 1.3576,Y -6.4774,Z 20,A -2.9828,B 0,C 0,E1 0.1598,E2 90.0716} C_DIS
LIN {X 2.0808,Y -6.2813,Z 20,A -2.948,B 0,C 0,E1 0.1598,E2 90.0716} C_DIS
LIN {X 2.7782,Y -6.0073,Z 20,A -2.9108,B 0,C 0,E1 0.1598,E2 90.0716} C_DIS
LIN {X 3.4393,Y -5.6544,Z 20,A -2.8715,B 0,C 0,E1 0.1598,E2 90.0716} C_DIS
LIN {X 4.0565,Y -5.2293,Z 20,A -2.8308,B 0,C 0,E1 0.1598,E2 90.0717} C_DIS
LIN {X 4.6225,Y -4.7381,Z 20,A -2.7891,B 0,C 0,E1 0.1598,E2 90.0717} C_DIS
LIN {X 5.129,Y -4.1856,Z 20,A -2.747,B 0,C 0,E1 0.1598,E2 90.0717} C_DIS
LIN {X 5.5694,Y -3.5793,Z 20,A -2.705,B 0,C 0,E1 0.1598,E2 90.0717} C_DIS
LIN {X 5.9379,Y -2.9266,Z 20,A -2.6637,B 0,C 0,E1 0.1598,E2 90.0717} C_DIS
LIN {X 6.231,Y -2.237,Z 20,A -2.6235,B 0,C 0,E1 0.1598,E2 90.0718} C_DIS
LIN {X 6.4434,Y -1.5182,Z 20,A -2.5851,B 0,C 0,E1 0.1598,E2 90.0718} C_DIS
LIN {X 6.5719,Y -0.7798,Z 20,A -2.549,B 0,C 0,E1 0.1598,E2 90.0718} C_DIS
LIN {X 6.6202,Y -0.032,Z 20,A -2.5154,B 0,C 0,E1 0.1598,E2 90.0719} C_DIS
LIN {X 6.5804,Y 0.7164,Z 20,A -2.4851,B 0,C 0,E1 0.1598,E2 90.0719} C_DIS
LIN {X 6.4552,Y 1.4553,Z 20,A -2.4583,B 0,C 0,E1 0.1598,E2 90.0719} C_DIS
LIN {X 6.2506,Y 2.1761,Z 20,A -2.4352,B 0,C 0,E1 0.1598,E2 90.072} C_DIS
LIN {X 5.9644,Y 2.8687,Z 20,A -2.4164,B 0,C 0,E1 0.1598,E2 90.072} C_DIS
LIN {X 5.6019,Y 3.5246,Z 20,A -2.4019,B 0,C 0,E1 0.1598,E2 90.0721} C_DIS
LIN {X 5.1684,Y 4.1359,Z 20,A -2.392,B 0,C 0,E1 0.1598,E2 90.0721} C_DIS
LIN {X 4.6671,Y 4.6931,Z 20,A -2.3869,B 0,C 0,E1 0.1598,E2 90.0722} C_DIS
LIN {X 4.1059,Y 5.1896,Z 20,A -2.3865,B 0,C 0,E1 0.1598,E2 90.0722} C_DIS
LIN {X 3.4932,Y 5.621,Z 20,A -2.3909,B 0,C 0,E1 0.1598,E2 90.0722} C_DIS
LIN {X 2.835,Y 5.979,Z 20,A -2.4,B 0,C 0,E1 0.1598,E2 90.0722} C_DIS
LIN {X 2.1417,Y 6.2637,Z 20,A -2.4136,B 0,C 0,E1 0.1598,E2 90.0722} C_DIS
LIN {X 1.1075,Y 6.5302,Z 20,A -2.4405,B 0,C 0,E1 0.1598,E2 90.0722} C_DIS
LIN {X 0.1968,Y 6.6156,Z 20,A -2.4705,B 0,C 0,E1 0.1598,E2 90.0722} C_DIS
LIN {X -0.5347,Y 6.5976,Z 20,A -2.4983,B 0,C 0,E1 0.1598,E2 90.0722} C_DIS
LIN {X -1.2598,Y 6.5,Z 20,A -2.5292,B 0,C 0,E1 0.1598,E2 90.0722} C_DIS
LIN {X -1.9696,Y 6.3223,Z 20,A -2.5628,B 0,C 0,E1 0.1598,E2 90.0722} C_DIS
LIN {X -2.6547,Y 6.0652,Z 20,A -2.599,B 0,C 0,E1 0.1598,E2 90.0721} C_DIS
LIN {X -3.3075,Y 5.7342,Z 20,A -2.637,B 0,C 0,E1 0.1598,E2 90.0721} C_DIS
LIN {X -3.9206,Y 5.3346,Z 20,A -2.6764,B 0,C 0,E1 0.1598,E2 90.0719} C_DIS
LIN {X -4.4855,Y 4.8696,Z 20,A -2.7168,B 0,C 0,E1 0.1598,E2 90.0719} C_DIS
LIN {X -4.9933,Y 4.3428,Z 20,A -2.7577,B 0,C 0,E1 0.1598,E2 90.0718} C_DIS
LIN {X -5.4421,Y 3.7651,Z 20,A -2.7986,B 0,C 0,E1 0.1598,E2 90.0717} C_DIS
LIN {X -5.826,Y 3.1422,Z 20,A -2.839,B 0,C 0,E1 0.1598,E2 90.0716} C_DIS
LIN {X -6.1375,Y 2.4803,Z 20,A -2.8784,B 0,C 0,E1 0.1598,E2 90.0716} C_DIS
LIN {X -6.3733,Y 1.7876,Z 20,A -2.9162,B 0,C 0,E1 0.1598,E2 90.0714} C_DIS
LIN {X -6.5315,Y 1.0731,Z 20,A -2.9522,B 0,C 0,E1 0.1598,E2 90.0714} C_DIS
LIN {X -6.6114,Y 0.3459,Z 20,A -2.9858,B 0,C 0,E1 0.1598,E2 90.0714} C_DIS
LIN {X -6.6075,Y -0.3858,Z 20,A -3.0165,B 0,C 0,E1 0.1598,E2 90.0713} C_DIS
LIN {X -6.5265,Y -1.113,Z 20,A -3.0442,B 0,C 0,E1 0.1598,E2 90.0713} C_DIS
LIN {X -6.3612,Y -1.8259,Z 20,A -3.0682,B 0,C 0,E1 0.1598,E2 90.0713} C_DIS
LIN {X -6.121,Y -2.517,Z 20,A -3.0886,B 0,C 0,E1 0.1598,E2 90.0713} C_DIS
LIN {X -5.8054,Y -3.1771,Z 20,A -3.1049,B 0,C 0,E1 0.1598,E2 90.0713} C_DIS
LIN {X -5.42,Y -3.7991,Z 20,A -3.117,B 0,C 0,E1 0.1598,E2 90.0713} C_DIS
LIN {X -4.9676,Y -4.3742,Z 20,A -3.1247,B 0,C 0,E1 0.1598,E2 90.0713} C_DIS
LIN {X -4.455,Y -4.8964,Z 20,A -3.128,B 0,C 0,E1 0.1598,E2 90.0713} C_DIS
LIN {X -3.8874,Y -5.3585,Z 20,A -3.1267,B 0,C 0,E1 0.1598,E2 90.0713} C_DIS
LIN {X -3.2712,Y -5.7531,Z 20,A -3.1209,B 0,C 0,E1 0.1598,E2 90.0713} C_DIS
LIN {X -2.6161,Y -6.0788,Z 20,A -3.1106,B 0,C 0,E1 0.1598,E2 90.0713} C_DIS
LIN {X -1.9298,Y -6.3325,Z 20,A -3.0962,B 0,C 0,E1 0.1598,E2 90.0714} C_DIS
LIN {X -1.2187,Y -6.5051,Z 20,A -3.0775,B 0,C 0,E1 0.1598,E2 90.0714} C_DIS
LIN {X -0.4933,Y -6.5997,Z 20,A -3.0549,B 0,C 0,E1 0.1598,E2 90.0714} C_DIS
LIN {X -0.4933,Y -6.5997,Z 20,A -3.0549,B 0,C 0,E1 0.1598,E2 90.0714} C_DIS
Enddeposition()
LIN {X 0.0882,Y -7.555,Z 20,A -3.0731,B 0,C 0,E1 0.1598,E2 90.0703} C_DIS
Startdeposition()
$VEL.CP = VEL_PRINT
LIN {X -0.5371,Y -7.5378,Z 20,A -3.0964,B 0,C 0,E1 0.1598,E2 90.0714} C_DIS
LIN {X -1.4345,Y -7.4203,Z 20,A -3.1244,B 0,C 0,E1 0.1598,E2 90.0714} C_DIS
LIN {X -2.3824,Y -7.1725,Z 20,A -3.1486,B 0,C 0,E1 0.1598,E2 90.0714} C_DIS
LIN {X -3.4378,Y -6.7246,Z 20,A -3.1683,B 0,C 0,E1 0.1598,E2 90.0712} C_DIS
LIN {X -4.1352,Y -6.3203,Z 20,A -3.1768,B 0,C 0,E1 0.1598,E2 90.0712} C_DIS
LIN {X -4.7853,Y -5.8436,Z 20,A -3.1804,B 0,C 0,E1 0.1598,E2 90.0712} C_DIS
LIN {X -5.3807,Y -5.3003,Z 20,A -3.1793,B 0,C 0,E1 0.1598,E2 90.0712} C_DIS
LIN {X -5.9152,Y -4.6969,Z 20,A -3.1733,B 0,C 0,E1 0.1598,E2 90.0712} C_DIS
LIN {X -6.5513,Y -3.7685,Z 20,A -3.1572,B 0,C 0,E1 0.1598,E2 90.0709} C_DIS
LIN {X -7.0411,Y -2.7337,Z 20,A -3.1315,B 0,C 0,E1 0.1598,E2 90.0709} C_DIS
LIN {X -7.386,Y -1.5981,Z 20,A -3.0961,B 0,C 0,E1 0.1598,E2 90.0709} C_DIS
LIN {X -7.5287,Y -0.6717,Z 20,A -3.0625,B 0,C 0,E1 0.1598,E2 90.0711} C_DIS
LIN {X -7.5527,Y 0.2738,Z 20,A -3.0235,B 0,C 0,E1 0.1598,E2 90.0711} C_DIS
LIN {X -7.418,Y 1.4217,Z 20,A -2.9698,B 0,C 0,E1 0.1598,E2 90.0709} C_DIS
LIN {X -7.0387,Y 2.7533,Z 20,A -2.8995,B 0,C 0,E1 0.1598,E2 90.0708} C_DIS
LIN {X -6.474,Y 3.8883,Z 20,A -2.8311,B 0,C 0,E1 0.1598,E2 90.0712} C_DIS
LIN {X -6.0408,Y 4.5334,Z 20,A -2.7884,B 0,C 0,E1 0.1598,E2 90.0716} C_DIS
LIN {X -5.2786,Y 5.408,Z 20,A -2.7233,B 0,C 0,E1 0.1598,E2 90.0716} C_DIS
LIN {X -4.5079,Y 6.0659,Z 20,A -2.6672,B 0,C 0,E1 0.1598,E2 90.0718} C_DIS
LIN {X -3.5665,Y 6.6581,Z 20,A -2.6076,B 0,C 0,E1 0.1598,E2 90.0719} C_DIS
LIN {X -2.7585,Y 7.0313,Z 20,A -2.5621,B 0,C 0,E1 0.1598,E2 90.0721} C_DIS
LIN {X -1.9126,Y 7.3075,Z 20,A -2.5193,B 0,C 0,E1 0.1598,E2 90.0721} C_DIS
LIN {X -0.651,Y 7.5302,Z 20,A -2.4633,B 0,C 0,E1 0.1598,E2 90.0723} C_DIS
LIN {X 0.3548,Y 7.5501,Z 20,A -2.4254,B 0,C 0,E1 0.1598,E2 90.0723} C_DIS
LIN {X 1.2909,Y 7.4463,Z 20,A -2.3952,B 0,C 0,E1 0.1598,E2 90.0723} C_DIS
LIN {X 2.3938,Y 7.1633,Z 20,A -2.3664,B 0,C 0,E1 0.1598,E2 90.0723} C_DIS
LIN {X 3.1407,Y 6.8684,Z 20,A -2.3513,B 0,C 0,E1 0.1598,E2 90.0723} C_DIS
LIN {X 3.8525,Y 6.4971,Z 20,A -2.3407,B 0,C 0,E1 0.1598,E2 90.0723} C_DIS
LIN {X 4.5208,Y 6.0519,Z 20,A -2.3349,B 0,C 0,E1 0.1598,E2 90.0723} C_DIS
LIN {X 5.1368,Y 5.5368,Z 20,A -2.334,B 0,C 0,E1 0.1598,E2 90.0723} C_DIS
LIN {X 5.932,Y 4.6818,Z 20,A -2.3407,B 0,C 0,E1 0.1598,E2 90.072} C_DIS
LIN {X 6.528,Y 3.7988,Z 20,A -2.3562,B 0,C 0,E1 0.1598,E2 90.072} C_DIS
LIN {X 7.0018,Y 2.8445,Z 20,A -2.3791,B 0,C 0,E1 0.1598,E2 90.0718} C_DIS
LIN {X 7.363,Y 1.6866,Z 20,A -2.4147,B 0,C 0,E1 0.1598,E2 90.0715} C_DIS
LIN {X 7.4958,Y 0.9657,Z 20,A -2.4409,B 0,C 0,E1 0.1598,E2 90.0719} C_DIS
LIN {X 7.557,Y -0.0807,Z 20,A -2.4829,B 0,C 0,E1 0.1598,E2 90.0716} C_DIS
LIN {X 7.4794,Y -1.0849,Z 20,A -2.5285,B 0,C 0,E1 0.1598,E2 90.0716} C_DIS
LIN {X 7.2333,Y -2.188,Z 20,A -2.5843,B 0,C 0,E1 0.1598,E2 90.0714} C_DIS
LIN {X 6.7426,Y -3.4139,Z 20,A -2.6544,B 0,C 0,E1 0.1598,E2 90.0713} C_DIS
LIN {X 6.2665,Y -4.2235,Z 20,A -2.7068,B 0,C 0,E1 0.1598,E2 90.0716} C_DIS
LIN {X 5.5136,Y -5.164,Z 20,A -2.7743,B 0,C 0,E1 0.1598,E2 90.0715} C_DIS
LIN {X 4.9704,Y -5.6873,Z 20,A -2.8168,B 0,C 0,E1 0.1598,E2 90.0717} C_DIS
LIN {X 4.3784,Y -6.1551,Z 20,A -2.8584,B 0,C 0,E1 0.1598,E2 90.0717} C_DIS
LIN {X 3.4586,Y -6.7208,Z 20,A -2.9162,B 0,C 0,E1 0.1598,E2 90.0715} C_DIS
LIN {X 2.4257,Y -7.153,Z 20,A -2.9725,B 0,C 0,E1 0.1598,E2 90.0715} C_DIS
LIN {X 1.4512,Y -7.4168,Z 20,A -3.0195,B 0,C 0,E1 0.1598,E2 90.0715} C_DIS
LIN {X 0.2932,Y -7.5477,Z 20,A -3.0675,B 0,C 0,E1 0.1598,E2 90.0715} C_DIS
LIN {X 0.2932,Y -7.5477,Z 20,A -3.0675,B 0,C 0,E1 0.1598,E2 90.0715} C_DIS
Enddeposition()
LIN {X 0.113,Y -8.4894,Z 20,A -3.1131,B 0,C 0,E1 0.1598,E2 90.0703} C_DIS
Startdeposition()
$VEL.CP = VEL_PRINT
LIN {X 1.1537,Y -8.4077,Z 20,A -3.0726,B 0,C 0,E1 0.1598,E2 90.0714} C_DIS
LIN {X 1.9744,Y -8.2533,Z 20,A -3.036,B 0,C 0,E1 0.1598,E2 90.0715} C_DIS
LIN {X 2.7761,Y -8.0191,Z 20,A -2.9967,B 0,C 0,E1 0.1598,E2 90.0715} C_DIS
LIN {X 3.5509,Y -7.7075,Z 20,A -2.955,B 0,C 0,E1 0.1598,E2 90.0715} C_DIS
LIN {X 4.2914,Y -7.3212,Z 20,A -2.9114,B 0,C 0,E1 0.1598,E2 90.0716} C_DIS
LIN {X 4.9904,Y -6.8642,Z 20,A -2.8663,B 0,C 0,E1 0.1598,E2 90.0716} C_DIS
LIN {X 5.6413,Y -6.3408,Z 20,A -2.8201,B 0,C 0,E1 0.1598,E2 90.0716} C_DIS
LIN {X 6.2379,Y -5.7561,Z 20,A -2.7733,B 0,C 0,E1 0.1598,E2 90.0717} C_DIS
LIN {X 6.9811,Y -4.8317,Z 20,A -2.7065,B 0,C 0,E1 0.1598,E2 90.0715} C_DIS
LIN {X 7.5242,Y -3.9256,Z 20,A -2.648,B 0,C 0,E1 0.1598,E2 90.0716} C_DIS
LIN {X 7.8777,Y -3.1578,Z 20,A -2.6024,B 0,C 0,E1 0.1598,E2 90.0718} C_DIS
LIN {X 8.1523,Y -2.3585,Z 20,A -2.5583,B 0,C 0,E1 0.1598,E2 90.0718} C_DIS
LIN {X 8.3459,Y -1.5358,Z 20,A -2.5161,B 0,C 0,E1 0.1598,E2 90.0718} C_DIS
LIN {X 8.4769,Y -0.4873,Z 20,A -2.4663,B 0,C 0,E1 0.1598,E2 90.0716} C_DIS
LIN {X 8.4599,Y 0.6845,Z 20,A -2.417,B 0,C 0,E1 0.1598,E2 90.0716} C_DIS
LIN {X 8.3509,Y 1.5141,Z 20,A -2.3861,B 0,C 0,E1 0.1598,E2 90.072} C_DIS
LIN {X 8.1612,Y 2.329,Z 20,A -2.3585,B 0,C 0,E1 0.1598,E2 90.072} C_DIS
LIN {X 7.8922,Y 3.1213,Z 20,A -2.3347,B 0,C 0,E1 0.1598,E2 90.072} C_DIS
LIN {X 7.5466,Y 3.8834,Z 20,A -2.3151,B 0,C 0,E1 0.1598,E2 90.0721} C_DIS
LIN {X 7.1277,Y 4.6077,Z 20,A -2.2998,B 0,C 0,E1 0.1598,E2 90.0721} C_DIS
LIN {X 6.6396,Y 5.2874,Z 20,A -2.289,B 0,C 0,E1 0.1598,E2 90.0722} C_DIS
LIN {X 5.9413,Y 6.0661,Z 20,A -2.2815,B 0,C 0,E1 0.1598,E2 90.0722} C_DIS
LIN {X 5.0524,Y 6.8196,Z 20,A -2.2824,B 0,C 0,E1 0.1598,E2 90.0722} C_DIS
LIN {X 4.3671,Y 7.2782,Z 20,A -2.2885,B 0,C 0,E1 0.1598,E2 90.0724} C_DIS
LIN {X 3.6403,Y 7.6679,Z 20,A -2.2989,B 0,C 0,E1 0.1598,E2 90.0724} C_DIS
LIN {X 2.8792,Y 7.9853,Z 20,A -2.3136,B 0,C 0,E1 0.1598,E2 90.0724} C_DIS
LIN {X 2.0908,Y 8.2273,Z 20,A -2.3325,B 0,C 0,E1 0.1598,E2 90.0724} C_DIS
LIN {X 1.2826,Y 8.3913,Z 20,A -2.3554,B 0,C 0,E1 0.1598,E2 90.0724} C_DIS
LIN {X 0.462,Y 8.4746,Z 20,A -2.3822,B 0,C 0,E1 0.1598,E2 90.0724} C_DIS
LIN {X -0.3625,Y 8.4791,Z 20,A -2.4125,B 0,C 0,E1 0.1598,E2 90.0724} C_DIS
LIN {X -1.1836,Y 8.4032,Z 20,A -2.446,B 0,C 0,E1 0.1598,E2 90.0724} C_DIS
LIN {X -1.9936,Y 8.2485,Z 20,A -2.4824,B 0,C 0,E1 0.1598,E2 90.0723} C_DIS
LIN {X -2.7848,Y 8.0162,Z 20,A -2.5214,B 0,C 0,E1 0.1598,E2 90.0722} C_DIS
LIN {X -3.5498,Y 7.7083,Z 20,A -2.5626,B 0,C 0,E1 0.1598,E2 90.0722} C_DIS
LIN {X -4.2814,Y 7.3276,Z 20,A -2.6057,B 0,C 0,E1 0.1598,E2 90.072} C_DIS
LIN {X -4.9727,Y 6.8779,Z 20,A -2.6501,B 0,C 0,E1 0.1598,E2 90.072} C_DIS
LIN {X -5.6172,Y 6.3632,Z 20,A -2.6955,B 0,C 0,E1 0.1598,E2 90.0718} C_DIS
LIN {X -6.4352,Y 5.538,Z 20,A -2.7603,B 0,C 0,E1 0.1598,E2 90.0716} C_DIS
LIN {X -7.0364,Y 4.7468,Z 20,A -2.8158,B 0,C 0,E1 0.1598,E2 90.0716} C_DIS
LIN {X -7.4473,Y 4.0664,Z 20,A -2.8597,B 0,C 0,E1 0.1598,E2 90.0716} C_DIS
LIN {X -7.7954,Y 3.3518,Z 20,A -2.9026,B 0,C 0,E1 0.1598,E2 90.0714} C_DIS
LIN {X -8.0753,Y 2.6079,Z 20,A -2.9442,B 0,C 0,E1 0.1598,E2 90.0714} C_DIS
LIN {X -8.2853,Y 1.8412,Z 20,A -2.9842,B 0,C 0,E1 0.1598,E2 90.0713} C_DIS
LIN {X -8.4648,Y 0.6672,Z 20,A -3.0399,B 0,C 0,E1 0.1598,E2 90.0708} C_DIS
LIN {X -8.4907,Y -0.0884,Z 20,A -3.0729,B 0,C 0,E1 0.1598,E2 90.0711} C_DIS
LIN {X -8.4166,Y -1.0964,Z 20,A -3.1126,B 0,C 0,E1 0.1598,E2 90.071} C_DIS
LIN {X -8.2742,Y -1.8925,Z 20,A -3.1411,B 0,C 0,E1 0.1598,E2 90.071} C_DIS
LIN {X -8.0559,Y -2.6711,Z 20,A -3.1659,B 0,C 0,E1 0.1598,E2 90.071} C_DIS
LIN {X -7.7645,Y -3.4254,Z 20,A -3.1871,B 0,C 0,E1 0.1598,E2 90.071} C_DIS
LIN {X -7.4028,Y -4.1486,Z 20,A -3.2043,B 0,C 0,E1 0.1598,E2 90.071} C_DIS
LIN {X -6.9754,Y -4.835,Z 20,A -3.2176,B 0,C 0,E1 0.1598,E2 90.071} C_DIS
LIN {X -6.3543,Y -5.6325,Z 20,A -3.2284,B 0,C 0,E1 0.1598,E2 90.0709} C_DIS
LIN {X -5.5431,Y -6.4308,Z 20,A -3.2324,B 0,C 0,E1 0.1598,E2 90.0709} C_DIS
LIN {X -4.7273,Y -7.0492,Z 20,A -3.2288,B 0,C 0,E1 0.1598,E2 90.0711} C_DIS
LIN {X -4.0263,Y -7.4726,Z 20,A -3.2211,B 0,C 0,E1 0.1598,E2 90.0711} C_DIS
LIN {X -3.2878,Y -7.8264,Z 20,A -3.209,B 0,C 0,E1 0.1598,E2 90.0712} C_DIS
LIN {X -2.5184,Y -8.1073,Z 20,A -3.1927,B 0,C 0,E1 0.1598,E2 90.0712} C_DIS
LIN {X -1.5249,Y -8.3541,Z 20,A -3.1668,B 0,C 0,E1 0.1598,E2 90.0713} C_DIS
LIN {X -0.5648,Y -8.4717,Z 20,A -3.1366,B 0,C 0,E1 0.1598,E2 90.0713} C_DIS
LIN {X 0.113,Y -8.4894,Z 20,A -3.1125,B 0,C 0,E1 0.1598,E2 90.0714} C_DIS
Enddeposition()
LIN {X 0.0004,Y -4.7523,Z 21,A -2.943,B 0,C 0,E1 0.1598,E2 90.0603} C_DIS
Startdeposition()
$VEL.CP = VEL_PRINT
LIN {X 0.0004,Y -4.7523,Z 21,A -2.9487,B 0,C 0,E1 0.1598,E2 90.0661} C_DIS
LIN {X -0.7614,Y -4.687,Z 21,A -2.9788,B 0,C 0,E1 0.1598,E2 90.0709} C_DIS
LIN {X -1.3211,Y -4.5628,Z 21,A -2.9947,B 0,C 0,E1 0.1598,E2 90.0715} C_DIS
LIN {X -2.0354,Y -4.2907,Z 21,A -3.0094,B 0,C 0,E1 0.1598,E2 90.0715} C_DIS
LIN {X -2.6978,Y -3.9091,Z 21,A -3.0175,B 0,C 0,E1 0.1598,E2 90.0715} C_DIS
LIN {X -3.2905,Y -3.4264,Z 21,A -3.0188,B 0,C 0,E1 0.1598,E2 90.0715} C_DIS
LIN {X -3.7962,Y -2.8533,Z 21,A -3.0131,B 0,C 0,E1 0.1598,E2 90.0714} C_DIS
LIN {X -4.2054,Y -2.2076,Z 21,A -3.0008,B 0,C 0,E1 0.1598,E2 90.0714} C_DIS
LIN {X -4.5059,Y -1.5048,Z 21,A -2.9821,B 0,C 0,E1 0.1598,E2 90.0714} C_DIS
LIN {X -4.6892,Y -0.7625,Z 21,A -2.9574,B 0,C 0,E1 0.1598,E2 90.0714} C_DIS
LIN {X -4.7516,Y -0.0006,Z 21,A -2.9275,B 0,C 0,E1 0.1598,E2 90.0714} C_DIS
LIN {X -4.6902,Y 0.7617,Z 21,A -2.8931,B 0,C 0,E1 0.1598,E2 90.0714} C_DIS
LIN {X -4.4744,Y 1.5941,Z 21,A -2.8499,B 0,C 0,E1 0.1598,E2 90.0714} C_DIS
LIN {X -4.2058,Y 2.2069,Z 21,A -2.8143,B 0,C 0,E1 0.1598,E2 90.0716} C_DIS
LIN {X -3.7983,Y 2.8538,Z 21,A -2.772,B 0,C 0,E1 0.1598,E2 90.0716} C_DIS
LIN {X -3.2209,Y 3.4906,Z 21,A -2.7238,B 0,C 0,E1 0.1598,E2 90.0717} C_DIS
LIN {X -2.6984,Y 3.9083,Z 21,A -2.687,B 0,C 0,E1 0.1598,E2 90.0719} C_DIS
LIN {X -2.0363,Y 4.2903,Z 21,A -2.6465,B 0,C 0,E1 0.1598,E2 90.0719} C_DIS
LIN {X -1.3218,Y 4.5618,Z 21,A -2.6087,B 0,C 0,E1 0.1598,E2 90.0721} C_DIS
LIN {X -0.5731,Y 4.7169,Z 21,A -2.5746,B 0,C 0,E1 0.1598,E2 90.0721} C_DIS
LIN {X 0.1907,Y 4.7473,Z 21,A -2.5452,B 0,C 0,E1 0.1598,E2 90.0721} C_DIS
LIN {X 0.9497,Y 4.6548,Z 21,A -2.5211,B 0,C 0,E1 0.1598,E2 90.0722} C_DIS
LIN {X 1.684,Y 4.4421,Z 21,A -2.503,B 0,C 0,E1 0.1598,E2 90.0722} C_DIS
LIN {X 2.3754,Y 4.1155,Z 21,A -2.4913,B 0,C 0,E1 0.1598,E2 90.0722} C_DIS
LIN {X 3.0049,Y 3.6812,Z 21,A -2.4865,B 0,C 0,E1 0.1598,E2 90.0722} C_DIS
LIN {X 3.5563,Y 3.1512,Z 21,A -2.4886,B 0,C 0,E1 0.1598,E2 90.0721} C_DIS
LIN {X 4.0646,Y 2.4577,Z 21,A -2.4991,B 0,C 0,E1 0.1598,E2 90.0719} C_DIS
LIN {X 4.3697,Y 1.8622,Z 21,A -2.5132,B 0,C 0,E1 0.1598,E2 90.0719} C_DIS
LIN {X 4.6109,Y 1.1368,Z 21,A -2.535,B 0,C 0,E1 0.1598,E2 90.0719} C_DIS
LIN {X 4.7341,Y 0.3825,Z 21,A -2.5625,B 0,C 0,E1 0.1598,E2 90.0719} C_DIS
LIN {X 4.7347,Y -0.3818,Z 21,A -2.5949,B 0,C 0,E1 0.1598,E2 90.0718} C_DIS
LIN {X 4.6112,Y -1.1361,Z 21,A -2.6315,B 0,C 0,E1 0.1598,E2 90.0718} C_DIS
LIN {X 4.3696,Y -1.8613,Z 21,A -2.6712,B 0,C 0,E1 0.1598,E2 90.0718} C_DIS
LIN {X 4.0139,Y -2.5377,Z 21,A -2.7131,B 0,C 0,E1 0.1598,E2 90.0718} C_DIS
LIN {X 3.5547,Y -3.1485,Z 21,A -2.7559,B 0,C 0,E1 0.1598,E2 90.0718} C_DIS
LIN {X 3.0044,Y -3.679,Z 21,A -2.7987,B 0,C 0,E1 0.1598,E2 90.0718} C_DIS
LIN {X 2.3746,Y -4.1121,Z 21,A -2.8403,B 0,C 0,E1 0.1598,E2 90.0717} C_DIS
LIN {X 1.6842,Y -4.4398,Z 21,A -2.8796,B 0,C 0,E1 0.1598,E2 90.0717} C_DIS
LIN {X 0.9505,Y -4.6537,Z 21,A -2.9156,B 0,C 0,E1 0.1598,E2 90.0717} C_DIS
LIN {X 0.1916,Y -4.7449,Z 21,A -2.9473,B 0,C 0,E1 0.1598,E2 90.0717} C_DIS
LIN {X 0.1916,Y -4.7449,Z 21,A -2.9473,B 0,C 0,E1 0.1598,E2 90.0717} C_DIS
Enddeposition()
LIN {X -0.0253,Y -5.6869,Z 21,A -2.9942,B 0,C 0,E1 0.1598,E2 90.0704} C_DIS
Startdeposition()
$VEL.CP = VEL_PRINT
LIN {X 0.6033,Y -5.6511,Z 21,A -2.9707,B 0,C 0,E1 0.1598,E2 90.0716} C_DIS
LIN {X 1.4284,Y -5.4997,Z 21,A -2.9341,B 0,C 0,E1 0.1598,E2 90.0716} C_DIS
LIN {X 2.2224,Y -5.2291,Z 21,A -2.8934,B 0,C 0,E1 0.1598,E2 90.0716} C_DIS
LIN {X 2.9681,Y -4.8451,Z 21,A -2.8497,B 0,C 0,E1 0.1598,E2 90.0717} C_DIS
LIN {X 3.6486,Y -4.3547,Z 21,A -2.8039,B 0,C 0,E1 0.1598,E2 90.0717} C_DIS
LIN {X 4.2506,Y -3.7708,Z 21,A -2.7569,B 0,C 0,E1 0.1598,E2 90.0717} C_DIS
LIN {X 4.7594,Y -3.1038,Z 21,A -2.7098,B 0,C 0,E1 0.1598,E2 90.0717} C_DIS
LIN {X 5.1649,Y -2.3696,Z 21,A -2.6636,B 0,C 0,E1 0.1598,E2 90.0717} C_DIS
LIN {X 5.4575,Y -1.5834,Z 21,A -2.6194,B 0,C 0,E1 0.1598,E2 90.0717} C_DIS
LIN {X 5.6309,Y -0.7627,Z 21,A -2.5781,B 0,C 0,E1 0.1598,E2 90.0717} C_DIS
LIN {X 5.682,Y 0.0745,Z 21,A -2.5407,B 0,C 0,E1 0.1598,E2 90.0717} C_DIS
LIN {X 5.6089,Y 0.9101,Z 21,A -2.5078,B 0,C 0,E1 0.1598,E2 90.0718} C_DIS
LIN {X 5.4143,Y 1.7261,Z 21,A -2.4804,B 0,C 0,E1 0.1598,E2 90.0718} C_DIS
LIN {X 5.1006,Y 2.504,Z 21,A -2.4589,B 0,C 0,E1 0.1598,E2 90.0719} C_DIS
LIN {X 4.6765,Y 3.2277,Z 21,A -2.4439,B 0,C 0,E1 0.1598,E2 90.072} C_DIS
LIN {X 4.1501,Y 3.8807,Z 21,A -2.4356,B 0,C 0,E1 0.1598,E2 90.072} C_DIS
LIN {X 3.5336,Y 4.4495,Z 21,A -2.4343,B 0,C 0,E1 0.1598,E2 90.0721} C_DIS
LIN {X 2.8403,Y 4.9216,Z 21,A -2.4399,B 0,C 0,E1 0.1598,E2 90.0721} C_DIS
LIN {X 2.0848,Y 5.2862,Z 21,A -2.4524,B 0,C 0,E1 0.1598,E2 90.0722} C_DIS
LIN {X 1.2842,Y 5.5368,Z 21,A -2.4713,B 0,C 0,E1 0.1598,E2 90.0722} C_DIS
LIN {X 0.4552,Y 5.6669,Z 21,A -2.4964,B 0,C 0,E1 0.1598,E2 90.0722} C_DIS
LIN {X -0.384,Y 5.6724,Z 21,A -2.5272,B 0,C 0,E1 0.1598,E2 90.0722} C_DIS
LIN {X -1.2146,Y 5.5526,Z 21,A -2.5629,B 0,C 0,E1 0.1598,E2 90.0722} C_DIS
LIN {X -1.8233,Y 5.3902,Z 21,A -2.5922,B 0,C 0,E1 0.1598,E2 90.0722} C_DIS
LIN {X -3.0679,Y 4.7921,Z 21,A -2.6631,B 0,C 0,E1 0.1598,E2 90.0718} C_DIS
LIN {X -3.8076,Y 4.2202,Z 21,A -2.7146,B 0,C 0,E1 0.1598,E2 90.0718} C_DIS
LIN {X -4.3281,Y 3.6832,Z 21,A -2.7564,B 0,C 0,E1 0.1598,E2 90.0718} C_DIS
LIN {X -4.7742,Y 3.083,Z 21,A -2.7982,B 0,C 0,E1 0.1598,E2 90.0717} C_DIS
LIN {X -5.1384,Y 2.4298,Z 21,A -2.8391,B 0,C 0,E1 0.1598,E2 90.0716} C_DIS
LIN {X -5.4141,Y 1.7345,Z 21,A -2.8786,B 0,C 0,E1 0.1598,E2 90.0715} C_DIS
LIN {X -5.5954,Y 1.0087,Z 21,A -2.9158,B 0,C 0,E1 0.1598,E2 90.0715} C_DIS
LIN {X -5.679,Y 0.2653,Z 21,A -2.9503,B 0,C 0,E1 0.1598,E2 90.0714} C_DIS
LIN {X -5.6627,Y -0.4823,Z 21,A -2.9812,B 0,C 0,E1 0.1598,E2 90.0714} C_DIS
LIN {X -5.5515,Y -1.2219,Z 21,A -3.0084,B 0,C 0,E1 0.1598,E2 90.0713} C_DIS
LIN {X -5.3414,Y -1.9396,Z 21,A -3.031,B 0,C 0,E1 0.1598,E2 90.0713} C_DIS
LIN {X -5.0427,Y -2.6253,Z 21,A -3.049,B 0,C 0,E1 0.1598,E2 90.0713} C_DIS
LIN {X -4.655,Y -3.265,Z 21,A -3.0618,B 0,C 0,E1 0.1598,E2 90.0713} C_DIS
LIN {X -4.1838,Y -3.846,Z 21,A -3.0691,B 0,C 0,E1 0.1598,E2 90.0713} C_DIS
LIN {X -3.6432,Y -4.3629,Z 21,A -3.0711,B 0,C 0,E1 0.1598,E2 90.0713} C_DIS
LIN {X -3.0391,Y -4.8036,Z 21,A -3.0677,B 0,C 0,E1 0.1598,E2 90.0713} C_DIS
LIN {X -2.3815,Y -5.1598,Z 21,A -3.0586,B 0,C 0,E1 0.1598,E2 90.0714} C_DIS
LIN {X -1.6837,Y -5.4286,Z 21,A -3.0444,B 0,C 0,E1 0.1598,E2 90.0714} C_DIS
LIN {X -0.9566,Y -5.6048,Z 21,A -3.0252,B 0,C 0,E1 0.1598,E2 90.0715} C_DIS
LIN {X -0.0253,Y -5.6869,Z 21,A -2.9946,B 0,C 0,E1 0.1598,E2 90.0715} C_DIS
Enddeposition()
LIN {X -0.0253,Y -5.6869,Z 21,A -2.9946,B 0,C 0,E1 0.1598,E2 90.0715} C_DIS
Startdeposition()
$VEL.CP = VEL_PRINT
LIN {X -0.6274,Y -6.5901,Z 21,A -3.0545,B 0,C 0,E1 0.1598,E2 90.0709} C_DIS
LIN {X -1.3711,Y -6.4741,Z 21,A -3.0774,B 0,C 0,E1 0.1598,E2 90.0714} C_DIS
LIN {X -2.0974,Y -6.2765,Z 21,A -3.0957,B 0,C 0,E1 0.1598,E2 90.0714} C_DIS
LIN {X -2.7969,Y -5.9987,Z 21,A -3.1096,B 0,C 0,E1 0.1598,E2 90.0714} C_DIS
LIN {X -3.4602,Y -5.6427,Z 21,A -3.1188,B 0,C 0,E1 0.1598,E2 90.0714} C_DIS
LIN {X -4.0777,Y -5.2121,Z 21,A -3.1232,B 0,C 0,E1 0.1598,E2 90.0714} C_DIS
LIN {X -4.644,Y -4.7161,Z 21,A -3.123,B 0,C 0,E1 0.1598,E2 90.0713} C_DIS
LIN {X -5.1503,Y -4.159,Z 21,A -3.118,B 0,C 0,E1 0.1598,E2 90.0713} C_DIS
LIN {X -5.5883,Y -3.5467,Z 21,A -3.1082,B 0,C 0,E1 0.1598,E2 90.0713} C_DIS
LIN {X -5.9544,Y -2.8889,Z 21,A -3.0938,B 0,C 0,E1 0.1598,E2 90.0713} C_DIS
LIN {X -6.2431,Y -2.1938,Z 21,A -3.075,B 0,C 0,E1 0.1598,E2 90.0713} C_DIS
LIN {X -6.4538,Y -1.4711,Z 21,A -3.0523,B 0,C 0,E1 0.1598,E2 90.0713} C_DIS
LIN {X -6.5802,Y -0.7289,Z 21,A -3.0256,B 0,C 0,E1 0.1598,E2 90.0713} C_DIS
LIN {X -6.6195,Y 0.023,Z 21,A -2.9953,B 0,C 0,E1 0.1598,E2 90.0713} C_DIS
LIN {X -6.5751,Y 0.7743,Z 21,A -2.9619,B 0,C 0,E1 0.1598,E2 90.0713} C_DIS
LIN {X -6.444,Y 1.5158,Z 21,A -2.9258,B 0,C 0,E1 0.1598,E2 90.0713} C_DIS
LIN {X -6.2306,Y 2.2378,Z 21,A -2.8875,B 0,C 0,E1 0.1598,E2 90.0715} C_DIS
LIN {X -5.9369,Y 2.9309,Z 21,A -2.8475,B 0,C 0,E1 0.1598,E2 90.0715} C_DIS
LIN {X -5.5646,Y 3.5854,Z 21,A -2.8062,B 0,C 0,E1 0.1598,E2 90.0716} C_DIS
LIN {X -5.1216,Y 4.1942,Z 21,A -2.7642,B 0,C 0,E1 0.1598,E2 90.0717} C_DIS
LIN {X -4.6124,Y 4.7489,Z 21,A -2.7221,B 0,C 0,E1 0.1598,E2 90.0717} C_DIS
LIN {X -4.0446,Y 5.2432,Z 21,A -2.6803,B 0,C 0,E1 0.1598,E2 90.0719} C_DIS
LIN {X -3.4212,Y 5.6652,Z 21,A -2.6396,B 0,C 0,E1 0.1598,E2 90.0719} C_DIS
LIN {X -2.7559,Y 6.0174,Z 21,A -2.6002,B 0,C 0,E1 0.1598,E2 90.072} C_DIS
LIN {X -2.0557,Y 6.2936,Z 21,A -2.5627,B 0,C 0,E1 0.1598,E2 90.0721} C_DIS
LIN {X -1.328,Y 6.4862,Z 21,A -2.5277,B 0,C 0,E1 0.1598,E2 90.0721} C_DIS
LIN {X -0.5826,Y 6.5917,Z 21,A -2.4958,B 0,C 0,E1 0.1598,E2 90.0722} C_DIS
LIN {X 0.1697,Y 6.6164,Z 21,A -2.467,B 0,C 0,E1 0.1598,E2 90.0722} C_DIS
LIN {X 1.1068,Y 6.5303,Z 21,A -2.436,B 0,C 0,E1 0.1598,E2 90.0723} C_DIS
LIN {X 2.1346,Y 6.2662,Z 21,A -2.4093,B 0,C 0,E1 0.1598,E2 90.0723} C_DIS
LIN {X 2.8197,Y 5.9877,Z 21,A -2.3958,B 0,C 0,E1 0.1598,E2 90.0723} C_DIS
LIN {X 3.4699,Y 5.6353,Z 21,A -2.3867,B 0,C 0,E1 0.1598,E2 90.0723} C_DIS
LIN {X 4.0769,Y 5.213,Z 21,A -2.3822,B 0,C 0,E1 0.1598,E2 90.0723} C_DIS
LIN {X 4.633,Y 4.7255,Z 21,A -2.3823,B 0,C 0,E1 0.1598,E2 90.0723} C_DIS
LIN {X 5.1319,Y 4.1797,Z 21,A -2.387,B 0,C 0,E1 0.1598,E2 90.0723} C_DIS
LIN {X 5.5669,Y 3.5814,Z 21,A -2.3963,B 0,C 0,E1 0.1598,E2 90.0722} C_DIS
LIN {X 5.9313,Y 2.9378,Z 21,A -2.4102,B 0,C 0,E1 0.1598,E2 90.0722} C_DIS
LIN {X 6.2212,Y 2.2574,Z 21,A -2.4284,B 0,C 0,E1 0.1598,E2 90.0721} C_DIS
LIN {X 6.4345,Y 1.5493,Z 21,A -2.4506,B 0,C 0,E1 0.1598,E2 90.0721} C_DIS
LIN {X 6.5695,Y 0.822,Z 21,A -2.4765,B 0,C 0,E1 0.1598,E2 90.072} C_DIS
LIN {X 6.6176,Y 0.084,Z 21,A -2.5061,B 0,C 0,E1 0.1598,E2 90.072} C_DIS
LIN {X 6.5861,Y -0.6548,Z 21,A -2.5387,B 0,C 0,E1 0.1598,E2 90.0719} C_DIS
LIN {X 6.4722,Y -1.3855,Z 21,A -2.5739,B 0,C 0,E1 0.1598,E2 90.0719} C_DIS
LIN {X 6.2769,Y -2.0988,Z 21,A -2.6115,B 0,C 0,E1 0.1598,E2 90.0719} C_DIS
LIN {X 6.0054,Y -2.7867,Z 21,A -2.6507,B 0,C 0,E1 0.1598,E2 90.0718} C_DIS
LIN {X 5.6575,Y -3.4395,Z 21,A -2.6913,B 0,C 0,E1 0.1598,E2 90.0718} C_DIS
LIN {X 5.238,Y -4.0485,Z 21,A -2.7326,B 0,C 0,E1 0.1598,E2 90.0718} C_DIS
LIN {X 4.7521,Y -4.6063,Z 21,A -2.7742,B 0,C 0,E1 0.1598,E2 90.0718} C_DIS
LIN {X 4.209,Y -5.1082,Z 21,A -2.8155,B 0,C 0,E1 0.1598,E2 90.0717} C_DIS
LIN {X 3.6131,Y -5.5464,Z 21,A -2.856,B 0,C 0,E1 0.1598,E2 90.0717} C_DIS
LIN {X 2.9718,Y -5.915,Z 21,A -2.8952,B 0,C 0,E1 0.1598,E2 90.0717} C_DIS
LIN {X 2.2931,Y -6.2089,Z 21,A -2.9326,B 0,C 0,E1 0.1598,E2 90.0717} C_DIS
LIN {X 1.5859,Y -6.4254,Z 21,A -2.9678,B 0,C 0,E1 0.1598,E2 90.0716} C_DIS
LIN {X 0.859,Y -6.5616,Z 21,A -3.0002,B 0,C 0,E1 0.1598,E2 90.0716} C_DIS
LIN {X -0.0633,Y -6.6229,Z 21,A -3.0367,B 0,C 0,E1 0.1598,E2 90.0716} C_DIS
Enddeposition()
LIN {X -0.0633,Y -6.6229,Z 21,A -3.0367,B 0,C 0,E1 0.1598,E2 90.0716} C_DIS
Startdeposition()
$VEL.CP = VEL_PRINT
LIN {X -0.0098,Y -7.5586,Z 21,A -3.074,B 0,C 0,E1 0.1598,E2 90.0709} C_DIS
LIN {X 1.1388,Y -7.4663,Z 21,A -3.0285,B 0,C 0,E1 0.1598,E2 90.0715} C_DIS
LIN {X 1.9785,Y -7.289,Z 21,A -2.9902,B 0,C 0,E1 0.1598,E2 90.0715} C_DIS
LIN {X 2.9925,Y -6.9389,Z 21,A -2.9381,B 0,C 0,E1 0.1598,E2 90.0715} C_DIS
LIN {X 3.9034,Y -6.4707,Z 21,A -2.8848,B 0,C 0,E1 0.1598,E2 90.0716} C_DIS
LIN {X 4.8789,Y -5.7704,Z 21,A -2.8191,B 0,C 0,E1 0.1598,E2 90.0716} C_DIS
LIN {X 5.6695,Y -4.9968,Z 21,A -2.7571,B 0,C 0,E1 0.1598,E2 90.0716} C_DIS
LIN {X 6.2967,Y -4.1798,Z 21,A -2.6992,B 0,C 0,E1 0.1598,E2 90.0716} C_DIS
LIN {X 6.7432,Y -3.4125,Z 21,A -2.6501,B 0,C 0,E1 0.1598,E2 90.0716} C_DIS
LIN {X 7.2324,Y -2.1909,Z 21,A -2.5798,B 0,C 0,E1 0.1598,E2 90.0713} C_DIS
LIN {X 7.4784,Y -1.091,Z 21,A -2.5241,B 0,C 0,E1 0.1598,E2 90.0716} C_DIS
LIN {X 7.5569,Y -0.0852,Z 21,A -2.4785,B 0,C 0,E1 0.1598,E2 90.0717} C_DIS
LIN {X 7.4964,Y 0.9599,Z 21,A -2.4363,B 0,C 0,E1 0.1598,E2 90.0717} C_DIS
LIN {X 7.2525,Y 2.1114,Z 21,A -2.3961,B 0,C 0,E1 0.1598,E2 90.0716} C_DIS
LIN {X 7.0038,Y 2.8398,Z 21,A -2.3746,B 0,C 0,E1 0.1598,E2 90.0719} C_DIS
LIN {X 6.5435,Y 3.7736,Z 21,A -2.3519,B 0,C 0,E1 0.1598,E2 90.0719} C_DIS
LIN {X 5.9111,Y 4.7089,Z 21,A -2.3355,B 0,C 0,E1 0.1598,E2 90.0719} C_DIS
LIN {X 5.1158,Y 5.5571,Z 21,A -2.3289,B 0,C 0,E1 0.1598,E2 90.072} C_DIS
LIN {X 4.5009,Y 6.0661,Z 21,A -2.3302,B 0,C 0,E1 0.1598,E2 90.0723} C_DIS
LIN {X 3.8357,Y 6.5073,Z 21,A -2.3361,B 0,C 0,E1 0.1598,E2 90.0723} C_DIS
LIN {X 3.1271,Y 6.8745,Z 21,A -2.3467,B 0,C 0,E1 0.1598,E2 90.0723} C_DIS
LIN {X 2.3842,Y 7.1663,Z 21,A -2.3618,B 0,C 0,E1 0.1598,E2 90.0723} C_DIS
LIN {X 1.2941,Y 7.4458,Z 21,A -2.3903,B 0,C 0,E1 0.1598,E2 90.0723} C_DIS
LIN {X 0.4164,Y 7.546,Z 21,A -2.4185,B 0,C 0,E1 0.1598,E2 90.0723} C_DIS
LIN {X -0.5889,Y 7.5344,Z 21,A -2.4561,B 0,C 0,E1 0.1598,E2 90.0723} C_DIS
LIN {X -1.7311,Y 7.3517,Z 21,A -2.5059,B 0,C 0,E1 0.1598,E2 90.0723} C_DIS
LIN {X -2.5165,Y 7.1197,Z 21,A -2.5447,B 0,C 0,E1 0.1598,E2 90.0722} C_DIS
LIN {X -3.2725,Y 6.8049,Z 21,A -2.5859,B 0,C 0,E1 0.1598,E2 90.0721} C_DIS
LIN {X -3.9916,Y 6.4128,Z 21,A -2.6289,B 0,C 0,E1 0.1598,E2 90.072} C_DIS
LIN {X -4.941,Y 5.7173,Z 21,A -2.6931,B 0,C 0,E1 0.1598,E2 90.0718} C_DIS
LIN {X -5.6758,Y 4.9894,Z 21,A -2.7508,B 0,C 0,E1 0.1598,E2 90.0716} C_DIS
LIN {X -6.2654,Y 4.2167,Z 21,A -2.8052,B 0,C 0,E1 0.1598,E2 90.0716} C_DIS
LIN {X -6.7592,Y 3.3796,Z 21,A -2.8585,B 0,C 0,E1 0.1598,E2 90.0713} C_DIS
LIN {X -7.2745,Y 2.0513,Z 21,A -2.933,B 0,C 0,E1 0.1598,E2 90.0708} C_DIS
LIN {X -7.47,Y 1.1432,Z 21,A -2.979,B 0,C 0,E1 0.1598,E2 90.0712} C_DIS
LIN {X -7.553,Y -0.0258,Z 21,A -3.0309,B 0,C 0,E1 0.1598,E2 90.0708} C_DIS
LIN {X -7.4558,Y -1.2318,Z 21,A -3.0783,B 0,C 0,E1 0.1598,E2 90.0708} C_DIS
LIN {X -7.1668,Y -2.3832,Z 21,A -3.1162,B 0,C 0,E1 0.1598,E2 90.0707} C_DIS
LIN {X -6.8497,Y -3.179,Z 21,A -3.1385,B 0,C 0,E1 0.1598,E2 90.071} C_DIS
LIN {X -6.4456,Y -3.934,Z 21,A -3.1556,B 0,C 0,E1 0.1598,E2 90.071} C_DIS
LIN {X -5.9585,Y -4.6385,Z 21,A -3.1675,B 0,C 0,E1 0.1598,E2 90.071} C_DIS
LIN {X -5.395,Y -5.2835,Z 21,A -3.1741,B 0,C 0,E1 0.1598,E2 90.0711} C_DIS
LIN {X -4.763,Y -5.8617,Z 21,A -3.1754,B 0,C 0,E1 0.1598,E2 90.0711} C_DIS
Enddeposition()
END
